	SwapInfo						:INT;
	VacValve_V8					:BOOL;	//白墨负压阀
	PurValve_V7					:BOOL;//正压阀
	alternate_Pumping		:BOOL;//交替加墨
	Swapping_Done			:BOOL;
	Error					:BOOL;
END_VAR
VAR
	step						:INT;
	stepA,stepB1,	stepB2		:INT;
	Ton,ton7,ton10				:TON;
	
	FB_SQUARE					:FB_SQUARE;
	W,X,A,Z,Y:INT;
	cycle_r_trig1,cycle_r_trig2  :R_TRIG;      //循坏
	cycle_x1,cycle_x2				:INT;//循坏次数
	purge_F_trig:F_TRIG;
	dely_off_setoff:TON;
	dely_emstop:Tc2_Standard.TON;
	ton1:Tc2_Standard.TON;
END_VAR
VAR_IN_OUT
	initialize				:BOOL;
	swap					:BOOL;
	CYCLE					:INT;//"0:Cycle A: Swap white ink to storage ;1:Cycle B: Swap storage to white ink"
	setoff					:BOOL;
END_VAR

IF setoff OR GVL.Reset THEN 
	step:=99;
END_IF
CASE step OF 
0://waiting
	IF initialize THEN 
		step :=5;
	ELSIF swap THEN 
		step :=10;
	ELSIF setoff OR GVL.Reset THEN 
		step :=99;
	END_IF
	
(***********当状态=Idle时，错误代码等于循坏错误****************************************)
	IF  state=MUStateEnum.idle THEN 
		error_code:=Circ_normal_error;
	END_IF
(***********自复位****************************************)	
	ton1(IN:=Swapping_Done , PT:= T#1S, Q=> , ET=> );
	IF ton1.Q THEN 
		Swapping_Done:=FALSE;
	END_IF
5://OFF
	state:=MUStateEnum.off;
	error_code:=MUErrorEnum.no_error;
	stepA:=stepB1:=stepB2:=0;
	W:=X:=A:=Z:=Y:=0;
	SwapInfo:=SwapInfoEnum.NONE;
	dely_emstop(IN:=FALSE);

	VacValve_V8:=FALSE;
	PurValve_V7:=FALSE;	
	
	GVL.fill_W_in_swap_enable:=FALSE;
	GVL.fill_F_in_swap_enable:=FALSE;
	
		IF initialize THEN //idle,此状态，所有泵停止	
			initialize:=FALSE;
			state:=MUStateEnum.idle;					
			GVL.fill_W_in_swap_enable:=FALSE;
			step:=0;
		END_IF
10://idle,此状态，所有泵停止				
		IF swap THEN 
			swap:=FALSE;
			state:=MUStateEnum.swapping;
			error_code:=MUErrorEnum.no_error;
			step:=20;
		END_IF
		
		IF error_code<>0 THEN 			
			step:=100;
		END_IF

20://SWAPPING		
		IF CYCLE=0 THEN
			ACT_Cycle_A();			
		ELSIF CYCLE=1 THEN 
			ACT_Cycle_B1();	
		END_IF
		
		IF SwapInfo=SwapInfoEnum.AC_STORAGE_FLUSH_FINISHED OR 
			SwapInfo=SwapInfoEnum.AC_WHITE_INK_FINISHED THEN 
			stepA:=stepB1:=stepB2:=0;		
			Swapping_Done:=TRUE;
			state:=MUStateEnum.idle;
			step:=0;
		END_IF
99://setoff
	setoff :=FALSE;
	error:=FALSE;
	state:=MUStateEnum.off;
	error_code:=MUErrorEnum.no_error;
	stepA:=stepB1:=stepB2:=0;
	W:=X:=A:=Z:=Y:=0;
	SwapInfo:=SwapInfoEnum.NONE;
	dely_emstop(IN:=FALSE);
	VacValve_V8:=FALSE;
	PurValve_V7:=FALSE;	
	
	GVL.fill_W_in_swap_enable:=FALSE;
	GVL.fill_F_in_swap_enable:=FALSE;
	step:=0;
100://error
		error:=TRUE;
		state:=MUStateEnum.error;
		stepA:=stepB1:=stepB2:=0;
		W:=X:=A:=Z:=Y:=0;
		dely_emstop(IN:=FALSE);
		VacValve_V8:=FALSE;
		PurValve_V7:=FALSE;	
		
		GVL.fill_W_in_swap_enable:=FALSE;
		GVL.fill_F_in_swap_enable:=FALSE;		
		step:=0;
END_CASE

IF setoff OR GVL.Reset THEN 
	step:=99;
END_IF

dely_off_setoff(IN:=setoff , PT:=T#1S , Q=> , ET=> );
IF dely_off_setoff.Q THEN
	setoff:=FALSE;
END_IF

IF state<>MUStateEnum.off AND state<>MUStateEnum.error  THEN 
	IF GVL.Emstop_Button THEN 
		error:=TRUE;
		error_code:=MUErrorEnum.emergency_error;
		PurValve_V7:=FALSE;
		dely_emstop(IN:=TRUE , PT:=T#1S , Q=> , ET=> );
		IF dely_emstop.Q THEN 
			VacValve_V8:=FALSE;
			step:=100;
		END_IF
	END_IF
END_IF

ACTION ACT_Cycle_A:
(***************Swap from White Ink to Storage Flush*******************************************)
CASE StepA OF
0:
	SwapInfo:=SwapInfoEnum.AC_STORAGE_FLUSH_RUNS;
	Ton(IN:=FALSE );	
	VacValve_V8:=FALSE;
	PurValve_V7 :=FALSE;
	stepA:=10;
10://SET "Vac White" OFF (valve 8 ON) 
	//START Pressure Purge Time = T1 (valve 7 ON)
	VacValve_V8:=TRUE;
	PurValve_V7 :=TRUE;
	Ton(IN:=TRUE , PT:=LREAL_TO_TIME(T[1]*1000) , Q=> , ET=> );
	IF Ton.Q THEN 
		Ton(IN:=FALSE );	
		stepA:=20;
	END_IF
20://STOP Pressure purge (normal filling conditions) (valve 7 OFF)	
	PurValve_V7:=FALSE;
	stepA:=30;
30://START Sol. filling (alternating pump time: T2=ON, T3=OFF)
	//WAIT UNTIL sensors in both TOP Sub Ink tanks detect a full tank (sensor 1 and 4)
	GVL.fill_F_in_swap_enable:=TRUE;
	alternate_Pumping:=TRUE;

	IF Sensor1 AND Sensor4 THEN 
		stepA:=31;
	END_IF
31://Wait Time: T4 (no vacuum)
	GVL.fill_F_in_swap_enable:=FALSE;
	alternate_Pumping:=FALSE;
	Ton(IN:=TRUE , PT:=LREAL_TO_TIME(T[4]*1000) , Q=> , ET=> );
		IF Ton.Q THEN 
			Ton(IN:=FALSE );
			stepA:=40;
		END_IF
40://Set "Vac White" ON  (Valve 8 OFF)     
	//Wait Time: T5 (filling conditions on & vac On)	
	VacValve_V8:=FALSE;	
	Ton(IN:=TRUE , PT:=LREAL_TO_TIME(T[5]*1000) , Q=> , ET=> );
	//调用加墨FB
		GVL.fill_F_in_swap_enable:=TRUE;
	IF Ton.Q THEN 
		stepA:=41;
	END_IF
41:
		GVL.fill_F_in_swap_enable:=FALSE;
		Ton(IN:=FALSE);
		stepA:=50;
50://Set "Vac White" Off (valve 8 ON)
	//For W=1 to 5 "Repeat 5x"
	//Pressure purge On for Time T6 (valve 7 ON)
	//Pressure purge Off for Time T6 (valve 7 OFF)
	VacValve_V8:=TRUE;
	FB_SQUARE(T_ON:=T[6] , T_OFF:=T[6] , SQUARE=>PurValve_V7 );
	purge_F_trig(CLK:=PurValve_V7 , Q=> );
	IF purge_F_trig.Q THEN 
		W:=W+1;
	END_IF
	
	IF W=6  THEN
		W:=0; 
		stepA:=60;
	END_IF
60://Wait  Time: T7 (while filling is ON)	
	Ton(IN:=TRUE  , PT:= LREAL_TO_TIME(T[7]*1000), Q=> , ET=> );	
	//调用加墨FB
	GVL.fill_F_in_swap_enable:=TRUE;
	IF ton.Q THEN 
		stepA:=61;
	END_IF
61:
		GVL.fill_F_in_swap_enable:=FALSE;
		Ton(IN:=FALSE);
		stepA:=70;
70://Set "Vac White" ON  (Valve 8 OFF)     
	//Wait Time: T5 (filling conditions on & vac On)
	VacValve_V8:=FALSE;
	//调用加墨FB
	GVL.fill_F_in_swap_enable:=TRUE;
	Ton(IN:=TRUE  , PT:= LREAL_TO_TIME(T[5]*1000), Q=> , ET=> );	
	IF ton.Q THEN 
		stepA:=71;
	END_IF
71:
		GVL.fill_F_in_swap_enable:=FALSE;
		Ton(IN:=FALSE);
		stepA:=80;
80://Set "Vac White" Off (valve 8 ON)
	VacValve_V8:=TRUE;
	//For X=1 to 5 "Repeat 5x"
	//Pressure purge On for Time T6 (valve 7 ON)
	//Pressure purge Off for Time T6 (valve 7 OFF)
	FB_SQUARE(T_ON:=T[6] , T_OFF:=T[6] , SQUARE=>PurValve_V7 );
	purge_F_trig(CLK:=PurValve_V7 , Q=> );
	IF purge_F_trig.Q THEN 
		X:=X+1;
	END_IF
	IF X=6  THEN 
		X:=0;
		stepA:=89;
	END_IF
89:
	A:=A+1;	
	stepA:=90;
90://Wait  Time: T7 (while filling is ON),第二次是T8	
	IF A<2 THEN 
		Ton(IN:=TRUE  , PT:= LREAL_TO_TIME(T[7]*1000), Q=> , ET=> );	
	ELSIF A=2 THEN 
		Ton(IN:=TRUE  , PT:= LREAL_TO_TIME(T[8]*1000), Q=> , ET=> );	
	END_IF
		//调用加墨FB
	GVL.fill_F_in_swap_enable:=TRUE;
	IF ton.Q THEN 
		stepA:=91;
	END_IF
91:
		GVL.fill_F_in_swap_enable:=FALSE;
		Ton(IN:=FALSE);
		stepA:=100;
100://Set "Vac White" ON  (Valve 8 OFF)    
	//Wait Time: T9 (filling conditions on) 
	VacValve_V8:=FALSE;
	//调用加墨FB
	GVL.fill_F_in_swap_enable:=TRUE;
	Ton(IN:=TRUE  , PT:= LREAL_TO_TIME(T[9]*1000), Q=> , ET=> );	
	IF ton.Q THEN 
		stepA:=101;
	END_IF	
101:
		GVL.fill_F_in_swap_enable:=FALSE;
		Ton(IN:=FALSE);
		stepA:=110;
110://重复	
	IF A<2 THEN 
		stepA:=10;
	ELSE stepA:=120;
	END_IF
120:(*FOR Z=1 to 5
	  IF both circulation pumps (3 & 6) were activated 3x within time: T13 => JUMP TO FINISH
	  ELSE Set Vac White Off (valve 8 ON)		
		NEXT Z*)
	A:=0;
	//	//调用加墨FB
	GVL.fill_F_in_swap_enable:=TRUE;
	Ton(IN:=TRUE  , PT:= LREAL_TO_TIME(T[13]*1000), Q=> , ET=> );	
	cycle_r_trig1(CLK:=Circ_Pump_L, Q=> );
	cycle_r_trig2(CLK:=Circ_Pump_R , Q=> );
		IF cycle_r_trig1.Q THEN 
			cycle_x1:=cycle_x1+1;
		END_IF
		IF cycle_r_trig2.Q THEN 
			cycle_x2:=cycle_x2+1;
		END_IF
		
	IF NOT Ton.Q AND cycle_x1>=3 AND cycle_x2>=3 THEN 
		Ton(IN:=FALSE);
		cycle_x1:=cycle_x2:=0;
		Z:=0;
		stepA:=190;
	ELSIF Ton.Q AND (cycle_x1<3 OR cycle_x2<3)  AND Z<5 THEN 	//循坏次数不够	
		Ton(IN:=FALSE);
		VacValve_V8:=TRUE;
		PurValve_V7:=TRUE;	
		cycle_x1:=cycle_x2:=0;
		stepA:=130;
	ELSIF Z=5 THEN
		Ton(IN:=FALSE);
		Z:=0; 
		stepA:=160;	
	END_IF
130://Start Pressure Purge On (valve 7 ON) for Time: T10
	//STOP Pressure purge (valve 7 OFF)   
			ton(IN:=TRUE , PT:= LREAL_TO_TIME(T[10]*1000) , Q=> , ET=> );		
			IF ton.Q THEN
				 ton(IN:=FALSE);
				PurValve_V7:=FALSE;
				stepA:=140;
			END_IF
140://Wait  Time: T7
		//Set "Vac White" ON  (Valve 8 OFF) 
			ton(IN:=TRUE , PT:= LREAL_TO_TIME(T[7]*1000) , Q=> , ET=> );
			IF Ton.Q THEN 
				ton(IN:=FALSE);
				VacValve_V8:=FALSE;		
				stepA:=150;
			END_IF
150://Wait Time: T11 (filling conditions on)
		//调用加墨FB
		ton(IN:=TRUE , PT:= LREAL_TO_TIME(T[11]*1000) , Q=> , ET=> );
			IF Ton.Q THEN 
				ton(IN:=FALSE);
				VacValve_V8:=FALSE;		
				Z:=Z+1;
				stepA:=120;
			END_IF
160://START WAIT = Message 2 on GUI 
	//If "PURGE BUTTON" is pushed during WAIT, THEN  
   //Set "Vac White" Off (valve 8 ON)
   //START Pressure purge (valve 7 ON) until button released
		SwapInfo:=SwapInfoEnum.AC_STORAGE_FLUSH_NEEDS_HELP;
			VacValve_V8:=TRUE;
		IF btPurge THEN 			
			PurValve_V7:=TRUE;
			stepA:=170;
		END_IF
170:    //START Pressure purge (valve 7 ON) until button released
		IF NOT btPurge THEN 
			PurValve_V7:=FALSE;
			stepA:=171;
		END_IF
171://Wait  Time: T7
	//Set "Vac White" ON  (Valve 8 OFF)  
		ton(IN:=TRUE , PT:= LREAL_TO_TIME(T[7]*1000) , Q=> , ET=> );
			IF Ton.Q THEN 
				ton(IN:=FALSE);
				VacValve_V8:=FALSE;
				stepA:=180;
			END_IF
180://  IF both circulation pumps (3 & 6) were activated 3x within time: T13 => JUMP TO FINISH
			//END IF (back TO wait)
		//	//调用加墨FB
	Ton(IN:=TRUE  , PT:= LREAL_TO_TIME(T[13]*1000), Q=> , ET=> );	
	cycle_r_trig1(CLK:=Circ_Pump_L, Q=> );
	cycle_r_trig2(CLK:=Circ_Pump_R , Q=> );
		IF cycle_r_trig1.Q THEN 
			cycle_x1:=cycle_x1+1;
		END_IF
		IF cycle_r_trig2.Q THEN 
			cycle_x2:=cycle_x2+1;
		END_IF
	IF NOT Ton.Q AND cycle_x1>=3 AND cycle_x2>=3 THEN 
		Ton(IN:=FALSE);
		cycle_x1:=cycle_x2:=0;
		stepA:=190;
	ELSIF Ton.Q AND (cycle_x1<3 OR cycle_x2<3) THEN 		
		Ton(IN:=FALSE);
		cycle_x1:=cycle_x2:=0;
		stepA:=160;
	END_IF
190:	//关闭所有供墨
	GVL.fill_F_in_swap_enable:=FALSE;
	stepA:=200;
200://FINISH => Message 3 on GUI
		SwapInfo:=SwapInfoEnum.AC_STORAGE_FLUSH_FINISHED;
		
END_CASE
END_ACTION

ACTION ACT_Cycle_B1:
(*************** Swap From Storage Flush to White Ink*******************************************)
CASE StepB1 OF
0:
	SwapInfo:=SwapInfoEnum.AC_WHITE_INK_RUNS;
	Ton(IN:=FALSE );	
	VacValve_V8:=FALSE;
	PurValve_V7 :=FALSE;
	StepB1:=10;
10://SET "Vac White" OFF (valve 8 ON) 
	//START Pressure Purge Time = T1 (valve 7 ON)
	VacValve_V8:=TRUE;
	PurValve_V7 :=TRUE;
	Ton(IN:=TRUE , PT:=LREAL_TO_TIME(T[1]*1000) , Q=> , ET=> );
	IF Ton.Q THEN 
		Ton(IN:=FALSE );	
		StepB1:=20;
	END_IF
20://STOP Pressure purge (normal filling conditions) (valve 7 OFF)	
	PurValve_V7:=FALSE;
	StepB1:=30;
30://START Ink filling  (alternating pump time: T2=ON, T3=OFF)
	//WAIT UNTIL sensors in both TOP Sub Ink tanks detect a full tank (sensor 1 and 4)	
	GVL.fill_W_in_swap_enable:=TRUE;
	alternate_Pumping:=TRUE;
	
	IF Sensor1 AND Sensor4 THEN 
		StepB1:=31;
	END_IF
31://Wait Time: T4 (no vacuum)
	GVL.fill_W_in_swap_enable:=FALSE;
	alternate_Pumping:=FALSE;
	Ton(IN:=TRUE , PT:=LREAL_TO_TIME(T[4]*1000) , Q=> , ET=> );
		IF Ton.Q THEN 
			Ton(IN:=FALSE );
			StepB1:=40;
		END_IF
40://Set "Vac White" ON  (Valve 8 OFF)     
	//Wait Time: T5 (filling conditions on & vac On)	
	VacValve_V8:=FALSE;	
	Ton(IN:=TRUE , PT:=LREAL_TO_TIME(T[5]*1000) , Q=> , ET=> );
	//调用加墨FB
		GVL.fill_W_in_swap_enable:=TRUE;
	IF Ton.Q THEN 
		StepB1:=41;
	END_IF
41:
		GVL.fill_W_in_swap_enable:=FALSE;
		Ton(IN:=FALSE);
		StepB1:=50;
50://Set "Vac White" Off (valve 8 ON)
	//For Z=1 to 5 "Repeat 5x"
	//Pressure purge On for Time T6 (valve 7 ON)
	//Pressure purge Off for Time T6 (valve 7 OFF)
	VacValve_V8:=TRUE;
	FB_SQUARE(T_ON:=T[6] , T_OFF:=T[6] , SQUARE=>PurValve_V7 );
	purge_F_trig(CLK:=PurValve_V7 , Q=> );
	IF purge_F_trig.Q THEN 
		Z:=Z+1;
	END_IF
	
	IF Z=6  THEN
		Z:=0; 
		StepB1:=60;
	END_IF
60://Wait  Time: T7
	Ton(IN:=TRUE  , PT:= LREAL_TO_TIME(T[7]*1000), Q=> , ET=> );	
	//调用加墨FB
	GVL.fill_W_in_swap_enable:=TRUE;
	IF ton.Q THEN 
		StepB1:=61;
	END_IF
61:
		GVL.fill_W_in_swap_enable:=FALSE;
		Ton(IN:=FALSE);
		StepB1:=70;
70://Set "Vac White" ON  (Valve 8 OFF)     
	//Wait Time: T5 (filling conditions on & vac On)
	VacValve_V8:=FALSE;
	//调用加墨FB
	GVL.fill_W_in_swap_enable:=TRUE;
	Ton(IN:=TRUE  , PT:= LREAL_TO_TIME(T[5]*1000), Q=> , ET=> );	
	IF ton.Q THEN 
		StepB1:=71;
	END_IF
71:
		GVL.fill_W_in_swap_enable:=FALSE;
		Ton(IN:=FALSE);
		StepB1:=80;
80://Set "Vac White" Off (valve 8 ON)
	VacValve_V8:=TRUE;
	//For Z=1 to 5 "Repeat 5x"
	//Pressure purge On for Time T6 (valve 7 ON)
	//Pressure purge Off for Time T6 (valve 7 OFF)
	FB_SQUARE(T_ON:=T[6] , T_OFF:=T[6] , SQUARE=>PurValve_V7 );
	purge_F_trig(CLK:=PurValve_V7 , Q=> );
	IF purge_F_trig.Q THEN 
		Z:=Z+1;
	END_IF
	IF Z=6  THEN 
		Z:=0;
		StepB1:=90;
	END_IF
90://Wait Time: T8 (filling conditions on, vac off))
		Ton(IN:=TRUE  , PT:= LREAL_TO_TIME(T[8]*1000), Q=> , ET=> );	
		//调用加墨FB
	GVL.fill_W_in_swap_enable:=TRUE;
	IF ton.Q THEN 
		StepB1:=91;
	END_IF
91:
		GVL.fill_W_in_swap_enable:=FALSE;
		Ton(IN:=FALSE);
		StepB1:=100;
100://Set "Vac White" ON  (Valve 8 OFF)    
	//Wait Time: T9 (filling conditions on) 
	VacValve_V8:=FALSE;
	//调用加墨FB
	GVL.fill_W_in_swap_enable:=TRUE;
	Ton(IN:=TRUE  , PT:= LREAL_TO_TIME(T[9]*1000), Q=> , ET=> );	
	IF ton.Q THEN 
		StepB1:=101;
	END_IF	
101:
		GVL.fill_W_in_swap_enable:=FALSE;
		Ton(IN:=FALSE);
		StepB1:=110;
110://无重复
		StepB1:=120;
120:(*FOR Y=1 to 5
	  IF both circulation pumps (3 & 6) were activated 3x within time: T13 => JUMP TO PAUSE
	  ELSE Set Vac White Off (valve 8 ON)		
		NEXT Y*)
	//	//调用加墨FB
	GVL.fill_W_in_swap_enable:=TRUE;
	Ton(IN:=TRUE  , PT:= LREAL_TO_TIME(T[13]*1000), Q=> , ET=> );	
	cycle_r_trig1(CLK:=Circ_Pump_L, Q=> );
	cycle_r_trig2(CLK:=Circ_Pump_R , Q=> );
		IF cycle_r_trig1.Q THEN 
			cycle_x1:=cycle_x1+1;
		END_IF
		IF cycle_r_trig2.Q THEN 
			cycle_x2:=cycle_x2+1;
		END_IF
		
	IF NOT Ton.Q AND cycle_x1>=3 AND cycle_x2>=3 THEN 
		Ton(IN:=FALSE);
		cycle_x1:=cycle_x2:=0;
		Y:=0;
		StepB1:=200;
	ELSIF Ton.Q AND (cycle_x1<3 OR cycle_x2<3)  AND Z<5 THEN 	//循坏次数不够,ELSE Set Vac White Off (valve 8 ON	
		Ton(IN:=FALSE);
		VacValve_V8:=TRUE;
		PurValve_V7:=TRUE;	
		cycle_x1:=cycle_x2:=0;
		StepB1:=130;
	ELSIF Y=5 THEN
		Ton(IN:=FALSE);
		Y:=0; 
		StepB1:=160;	
	END_IF
130://Start Pressure Purge On (valve 7 ON) for Time: T10
	//STOP Pressure purge (valve 7 OFF)   
			ton(IN:=TRUE , PT:= LREAL_TO_TIME(T[10]*1000) , Q=> , ET=> );		
			IF ton.Q THEN
				 ton(IN:=FALSE);
				PurValve_V7:=FALSE;
				StepB1:=140;
			END_IF
140://Wait  Time: T7
		//Set "Vac White" ON  (Valve 8 OFF) 
			ton(IN:=TRUE , PT:= LREAL_TO_TIME(T[7]*1000) , Q=> , ET=> );
			IF Ton.Q THEN 
				ton(IN:=FALSE);
				VacValve_V8:=FALSE;		
				StepB1:=150;
			END_IF
150://Wait Time: T11 (filling conditions on)
		//调用加墨FB
		ton(IN:=TRUE , PT:= LREAL_TO_TIME(T[11]*1000) , Q=> , ET=> );
			IF Ton.Q THEN 
				ton(IN:=FALSE);
				VacValve_V8:=FALSE;		
				Y:=Y+1;
				StepB1:=120;
			END_IF
160://START WAIT = Message 5 on GUI 
	//If "PURGE BUTTON" is pushed during WAIT, THEN  
   //Set "Vac White" Off (valve 8 ON)
   //START Pressure purge (valve 7 ON) until button released
		SwapInfo:=SwapInfoEnum.AC_WHITE_INK1_NEEDS_HELP;
			VacValve_V8:=TRUE;
		IF btPurge THEN 		
			PurValve_V7:=TRUE;
			StepB1:=170;
		END_IF
170:    //START Pressure purge (valve 7 ON) until button released
		IF NOT btPurge THEN 
			PurValve_V7:=FALSE;
			StepB1:=171;
		END_IF
171://Wait  Time: T7
	//Set "Vac White" ON  (Valve 8 OFF)  
		ton(IN:=TRUE , PT:= LREAL_TO_TIME(T[7]*1000) , Q=> , ET=> );
			IF Ton.Q THEN 
				ton(IN:=FALSE);
				VacValve_V8:=FALSE;
				StepB1:=180;
			END_IF
180://  IF both circulation pumps (3 & 6) were activated 3x within time T13 than:
		//           => remove Message 5
		//           => Show Message 4
		//           => JUMP TO PAUSE
		//END IF (back to wait)
				
		//	//调用加墨FB
	Ton(IN:=TRUE  , PT:= LREAL_TO_TIME(T[13]*1000), Q=> , ET=> );	
	cycle_r_trig1(CLK:=Circ_Pump_L, Q=> );
	cycle_r_trig2(CLK:=Circ_Pump_R , Q=> );
		IF cycle_r_trig1.Q THEN 
			cycle_x1:=cycle_x1+1;
		END_IF
		IF cycle_r_trig2.Q THEN 
			cycle_x2:=cycle_x2+1;
		END_IF
	IF NOT Ton.Q AND cycle_x1>=3 AND cycle_x2>=3 THEN 
		Ton(IN:=FALSE);
		cycle_x1:=cycle_x2:=0;
		StepB1:=190;
	ELSIF Ton.Q AND (cycle_x1<3 OR cycle_x2<3) THEN 		
		Ton(IN:=FALSE);
		cycle_x1:=cycle_x2:=0;
		StepB1:=160;
	END_IF
190:	//           => remove Message 5
		//           => Show Message 4
		//           => JUMP TO PAUSE
	SwapInfo:=SwapInfoEnum.AC_WHITE_INK_RUNS;	
	GVL.fill_W_in_swap_enable:=FALSE;
	StepB1:=200;
200://PAUSE:  wait time time: T12,Filter cleaning time
	//调用加墨FB
	GVL.fill_W_in_swap_enable:=TRUE;
	Ton(IN:=TRUE  , PT:= LREAL_TO_TIME(T[12]*1000), Q=> , ET=> );	
	IF Ton.Q THEN 
		StepB1:=210;		
	END_IF
210://关闭加墨
		Ton(IN:=FALSE);
		GVL.fill_W_in_swap_enable:=FALSE;
		StepB1:=220;
220://
	ACT_Cycle_B2();
		
END_CASE
END_ACTION

ACTION ACT_Cycle_B2:
(*************** Swap From Storage Flush to White Ink*******************************************)

CASE StepB2 OF
0:
	Ton(IN:=FALSE );	
	StepB2:=10;
10://SET "Vac White" OFF (valve 8 ON) 
	//START Pressure Purge Time = T1 (valve 7 ON)
	VacValve_V8:=TRUE;
	PurValve_V7 :=TRUE;
	Ton(IN:=TRUE , PT:=LREAL_TO_TIME(T[1]*1000) , Q=> , ET=> );
	IF Ton.Q THEN 
		Ton(IN:=FALSE );	
		StepB2:=20;
	END_IF
20://STOP Pressure purge (normal filling conditions) (valve 7 OFF)	
	PurValve_V7:=FALSE;
	StepB2:=30;
30://START Ink filling  (alternating pump time: T2=ON, T3=OFF)
	//WAIT UNTIL sensors in both TOP Sub Ink tanks detect a full tank (sensor 1 and 4)
	GVL.fill_W_in_swap_enable:=TRUE;
	alternate_Pumping:=TRUE;
	
	IF Sensor1 AND Sensor4 THEN 
		StepB2:=31;
	END_IF
31://Wait Time: T4 (no vacuum)
	GVL.fill_W_in_swap_enable:=FALSE;
	alternate_Pumping:=FALSE;
	Ton(IN:=TRUE , PT:=LREAL_TO_TIME(T[4]*1000) , Q=> , ET=> );
		IF Ton.Q THEN 
			Ton(IN:=FALSE );
			StepB2:=40;
		END_IF
40://Set "Vac White" ON  (Valve 8 OFF)     
	//Wait Time: T5 (filling conditions on & vac On)	
	VacValve_V8:=FALSE;	
	Ton(IN:=TRUE , PT:=LREAL_TO_TIME(T[5]*1000) , Q=> , ET=> );
	//调用加墨FB
		GVL.fill_W_in_swap_enable:=TRUE;
	IF Ton.Q THEN 
		StepB2:=41;
	END_IF
41:
		GVL.fill_W_in_swap_enable:=FALSE;
		Ton(IN:=FALSE);
		StepB2:=50;
50://Set "Vac White" Off (valve 8 ON)
	//For Z=1 to 5 "Repeat 5x"
	//Pressure purge On for Time T6 (valve 7 ON)
	//Pressure purge Off for Time T6 (valve 7 OFF)
	VacValve_V8:=TRUE;
	FB_SQUARE(T_ON:=T[6] , T_OFF:=T[6] , SQUARE=>PurValve_V7 );
	purge_F_trig(CLK:=PurValve_V7 , Q=> );
	IF purge_F_trig.Q THEN 
		Z:=Z+1;
	END_IF
	
	IF Z=6  THEN
		Z:=0; 
		StepB2:=60;
	END_IF
60://Wait  Time: T7
	Ton(IN:=TRUE  , PT:= LREAL_TO_TIME(T[7]*1000), Q=> , ET=> );	
	//调用加墨FB
	GVL.fill_W_in_swap_enable:=TRUE;
	IF ton.Q THEN 
		StepB2:=61;
	END_IF
61:
		GVL.fill_W_in_swap_enable:=FALSE;
		Ton(IN:=FALSE);
		StepB2:=70;
70://Set "Vac White" ON  (Valve 8 OFF)     
	//Wait Time: T5 (filling conditions on & vac On)
	VacValve_V8:=FALSE;
	//调用加墨FB
	GVL.fill_W_in_swap_enable:=TRUE;
	Ton(IN:=TRUE  , PT:= LREAL_TO_TIME(T[5]*1000), Q=> , ET=> );	
	IF ton.Q THEN 
		StepB2:=71;
	END_IF
71:
		GVL.fill_W_in_swap_enable:=FALSE;
		Ton(IN:=FALSE);
		StepB2:=80;
80://Set "Vac White" Off (valve 8 ON)
	VacValve_V8:=TRUE;
	//For Z=1 to 5 "Repeat 5x"
	//Pressure purge On for Time T6 (valve 7 ON)
	//Pressure purge Off for Time T6 (valve 7 OFF)
	FB_SQUARE(T_ON:=T[6] , T_OFF:=T[6] , SQUARE=>PurValve_V7 );
	purge_F_trig(CLK:=PurValve_V7 , Q=> );
	IF purge_F_trig.Q THEN 
		Z:=Z+1;
	END_IF
	IF Z=6  THEN 
		Z:=0;
		StepB2:=90;
	END_IF
90://Wait Time: T8 (filling conditions on, vac off))
		Ton(IN:=TRUE  , PT:= LREAL_TO_TIME(T[8]*1000), Q=> , ET=> );	
		//调用加墨FB
	GVL.fill_W_in_swap_enable:=TRUE;
	IF ton.Q THEN 
		StepB2:=91;
	END_IF
91:
		GVL.fill_W_in_swap_enable:=FALSE;
		Ton(IN:=FALSE);
		StepB2:=100;
100://Set "Vac White" ON  (Valve 8 OFF)    
	//Wait Time: T9 (filling conditions on) 
	VacValve_V8:=FALSE;
	//调用加墨FB
	GVL.fill_W_in_swap_enable:=TRUE;
	Ton(IN:=TRUE  , PT:= LREAL_TO_TIME(T[9]*1000), Q=> , ET=> );	
	IF ton.Q THEN 
		StepB2:=101;
	END_IF	
101:
		GVL.fill_W_in_swap_enable:=FALSE;
		Ton(IN:=FALSE);
		StepB2:=110;
110://无重复
		StepB2:=120;
120:(*FOR Z=1 to 5
	  IF both circulation pumps (3 & 6) were activated 3x within time: T13 => JUMP TO FINISH
	  ELSE Set Vac White Off (valve 8 ON)		
		NEXT Z*)
	//	//调用加墨FB
	GVL.fill_W_in_swap_enable:=TRUE;
	Ton(IN:=TRUE  , PT:= LREAL_TO_TIME(T[13]*1000), Q=> , ET=> );	
	cycle_r_trig1(CLK:=Circ_Pump_L, Q=> );
	cycle_r_trig2(CLK:=Circ_Pump_R , Q=> );
		IF cycle_r_trig1.Q THEN 
			cycle_x1:=cycle_x1+1;
		END_IF
		IF cycle_r_trig2.Q THEN 
			cycle_x2:=cycle_x2+1;
		END_IF
		
	IF NOT Ton.Q AND cycle_x1>=3 AND cycle_x2>=3 THEN 
		Ton(IN:=FALSE);
		cycle_x1:=cycle_x2:=0;
		Z:=0;
		StepB2:=200;
	ELSIF Ton.Q AND (cycle_x1<3 OR cycle_x2<3)  AND Z<5 THEN 	//循坏次数不够,ELSE Set Vac White Off (valve 8 ON	
		Ton(IN:=FALSE);
		VacValve_V8:=TRUE;
		PurValve_V7:=TRUE;	
		cycle_x1:=cycle_x2:=0;
		StepB2:=130;
	ELSIF Z=5 THEN
		Ton(IN:=FALSE);
		Z:=0; 
		StepB2:=160;	
	END_IF
130://Start Pressure Purge On (valve 7 ON) for Time: T10
	//STOP Pressure purge (valve 7 OFF)   
			ton(IN:=TRUE , PT:= LREAL_TO_TIME(T[10]*1000) , Q=> , ET=> );		
			IF ton.Q THEN
				 ton(IN:=FALSE);
				PurValve_V7:=FALSE;
				StepB2:=140;
			END_IF
140://Wait  Time: T7
		//Set "Vac White" ON  (Valve 8 OFF) 
			ton(IN:=TRUE , PT:= LREAL_TO_TIME(T[7]*1000) , Q=> , ET=> );
			IF Ton.Q THEN 
				ton(IN:=FALSE);
				VacValve_V8:=FALSE;		
				StepB2:=150;
			END_IF
150://Wait Time: T11 (filling conditions on)
		//调用加墨FB
		ton(IN:=TRUE , PT:= LREAL_TO_TIME(T[11]*1000) , Q=> , ET=> );
			IF Ton.Q THEN 
				ton(IN:=FALSE);
				VacValve_V8:=FALSE;		
				Z:=Z+1;
				StepB2:=120;
			END_IF
160://START WAIT = Message 6 on GUI 
	//If "PURGE BUTTON" is pushed during WAIT, THEN  
   //Set "Vac White" Off (valve 8 ON)
   //START Pressure purge (valve 7 ON) until button released
		SwapInfo:=SwapInfoEnum.AC_WHITE_INK2_NEEDS_HELP;
			VacValve_V8:=TRUE;
		IF btPurge THEN 			
			PurValve_V7:=TRUE;
			StepB2:=170;
		END_IF
170:    //START Pressure purge (valve 7 ON) until button released
		IF NOT btPurge THEN 
			PurValve_V7:=FALSE;
			StepB2:=171;
		END_IF
171://Wait  Time: T7
	//Set "Vac White" ON  (Valve 8 OFF)  
		ton(IN:=TRUE , PT:= LREAL_TO_TIME(T[7]*1000) , Q=> , ET=> );
			IF Ton.Q THEN 
				ton(IN:=FALSE);
				VacValve_V8:=FALSE;
				StepB2:=180;
			END_IF
180://    IF both circulation pumps (3 & 6) were activated 3x within time: T13 => JUMP TO FINISH
		//END IF (back to wait)
				
		//	//调用加墨FB
	Ton(IN:=TRUE  , PT:= LREAL_TO_TIME(T[13]*1000), Q=> , ET=> );	
	cycle_r_trig1(CLK:=Circ_Pump_L, Q=> );
	cycle_r_trig2(CLK:=Circ_Pump_R , Q=> );
		IF cycle_r_trig1.Q THEN 
			cycle_x1:=cycle_x1+1;
		END_IF
		IF cycle_r_trig2.Q THEN 
			cycle_x2:=cycle_x2+1;
		END_IF
	IF NOT Ton.Q AND cycle_x1>=3 AND cycle_x2>=3 THEN 
		Ton(IN:=FALSE);
		cycle_x1:=cycle_x2:=0;
		StepB2:=190;
	ELSIF Ton.Q AND (cycle_x1<3 OR cycle_x2<3) THEN 		
		Ton(IN:=FALSE);
		cycle_x1:=cycle_x2:=0;
		StepB2:=160;
	END_IF
190:	//  
	StepB2:=200;
200://
	StepB2:=210;
210://关闭加墨
	Ton(IN:=FALSE);
	GVL.fill_W_in_swap_enable:=FALSE;
	StepB2:=220;
220://FINISH => Message 7 on GUI
	SwapInfo:=SwapInfoEnum.AC_WHITE_INK_FINISHED;

		
END_CASE
END_ACTION

END_FUNCTION_BLOCK

// ---- POUs/MAIN.TcPOU
PROGRAM MAIN
VAR
	FB_count:FB_count;
END_VAR

P_UPS();
systime();

IO_Link();
P_API_IO();
P_Modbus();
MAIN_ALarm();

P_Motion();
P_MediaTransport();
P_System();
P_InkSystem();
P_UVLed();
P_RollToRoll();
P_SpitUnit();
P_MaintenanceUnit();
P_SubTank();
P_TwinSAFE();


ACT_heart();



//IF VisuElems.CURRENTVISU='VIS_AXIS' THEN 
	//VisuElems.CURRENTVISU:='VIS_ISS';
//END_IF

ACTION ACT_heart:
FB_count(Add_Time:=T#0.1S , count=> GVL_API.count );
END_ACTION

END_PROGRAM

// ---- POUs/040_System/P_System.TcPOU
PROGRAM P_System
VAR
END_VAR

P_FootPedal();
P_SystemEnvironment();
P_SafetyGuard();

END_PROGRAM

// ---- POUs/040_System/FootPedal/P_FootPedal.TcPOU
PROGRAM P_FootPedal
VAR
	FB_FootPedal:ARRAY[1..number_FootPedal] OF FB_FootPedal;//
	i:INT;
	log_ErrorEnum:FootPedalErrorEnum;
	log_ID:INT;
END_VAR

ACT_LOG();
FOR i:=1 TO number_FootPedal DO
	FB_FootPedal[i](
		PedalPressed1:=stInput.biFootPedal[i].PedalPressed1 , 
		PedalPressed2:=stInput.biFootPedal[i].PedalPressed2 , 
		PedalPressed3:=stInput.biFootPedal[i].PedalPressed3 , 
		debounce_time:=GVL_API.stFootPedal[i].debounce_time , 
		error_code=> GVL_API.stFootPedal[i].error_code, 
		state=> GVL_API.stFootPedal[i].state, 
		pressed=> GVL_API.stFootPedal[i].pressed, 
		Error=>GVL_API.stFootPedal[i].Error , 
		Reset:= GVL_API.stFootPedal[i].Reset );
END_FOR

ACTION ACT_LOG:
(*************************LOG*******************************************)
log_ID:=400;
FOR i:=1 TO number_FootPedal DO//401-404
//pressed
AlarmActionArray[log_ID+i].AlarmMsg.EN	:=CONCAT('FootPedal',
																			INT_TO_STRING(i));
AlarmActionArray[log_ID+i].AlarmMsg.EN	:=CONCAT(AlarmActionArray[log_ID+i].AlarmMsg.EN,': '	);																	
AlarmActionArray[log_ID+i].AlarmMsg.EN	:=CONCAT(AlarmActionArray[log_ID+i].AlarmMsg.EN,
																			INT_TO_STRING(GVL_API.stFootPedal[i].pressed));												
fbSetAlarm[log_ID+i](
	InUse:=TRUE , 
	EventId:=log_ID+i , 
	EventActive:=GVL_API.stFootPedal[i].pressed<>0 , 
	EventClass:=Alm_EventClass.Event , 
	ToTheLogFile:=TRUE, 
	ToTheHistory:=TRUE , 
 );
 
//ERROR,log_ErrorEnum只能等于一个常数,   410-414
CASE GVL_API.stUpDownSlot[i].error_code  OF
0	:	log_ErrorEnum	:=	0	;
1	:	log_ErrorEnum	:=	1	;
2	:	log_ErrorEnum	:=	2	;
3	:	log_ErrorEnum	:=	3	;
4	:	log_ErrorEnum	:=	4	;
666	:	log_ErrorEnum	:=	666	;


END_CASE
AlarmActionArray[log_ID+10+i].AlarmMsg.EN	:=CONCAT('FootPedal',INT_TO_STRING(i));
AlarmActionArray[log_ID+10+i].AlarmMsg.EN	:=CONCAT(AlarmActionArray[log_ID+10+i].AlarmMsg.EN,
																			' Error: ');
AlarmActionArray[log_ID+10+i].AlarmMsg.EN	:=CONCAT(AlarmActionArray[log_ID+10+i].AlarmMsg.EN,
																			TO_STRING(log_ErrorEnum));																			

fbSetAlarm[log_ID+10+i](
	InUse:=TRUE , 
	EventId:=log_ID+10+i , 
	EventActive:=GVL_API.stFootPedal[i].error_code<>0 AND GVL_API.stFootPedal[i].error_code<>666  , 
	EventClass:=Alm_EventClass.Alarm , 
	ToTheLogFile:=TRUE, 
	ToTheHistory:=TRUE , 
 );
 
//reset  420-424
AlarmActionArray[log_ID+20+i].AlarmMsg.EN	:=CONCAT('FootPedal',
																			INT_TO_STRING(i));
AlarmActionArray[log_ID+20+i].AlarmMsg.EN	:=CONCAT(AlarmActionArray[log_ID+20+i].AlarmMsg.EN,
																			' Reset');		

fbSetAlarm[log_ID+20+i](
	InUse:=TRUE , 
	EventId:=log_ID+20+i , 
	EventActive:=GVL_API.stFootPedal[i].Reset  , 
	EventClass:=Alm_EventClass.Event , 
	ToTheLogFile:=TRUE, 
	ToTheHistory:=TRUE , 
 );
END_FOR
END_ACTION

END_PROGRAM

// ---- POUs/060_UVLed/P_UVLed.TcPOU
PROGRAM P_UVLed
VAR
	//FB_UVLed		:FB_UVLed;
	FB_UVLed_L		:FB_UVLed_L;
	FB_UVLed_R		:FB_UVLed_R;

	log_ErrorEnum:UVLedErrorEnum;
	log_ID:INT;
	i:INT;
END_VAR

ACT_LOG();
FB_UVLed_L(
	single_double:=GVL_API.stUVLed[1].unidirection , 
	initial_print_position:= GVL_API.stUVLed[1].initial_print_position, 
	uv_power_leading:= GVL_API.stUVLed[1].uv_power_leading, 
	uv_power_trailing:= GVL_API.stUVLed[1].uv_power_trailing, 
	uvStart:= GVL_API.stUVLed[1].uvStart, 
	uvEnd:= GVL_API.stUVLed[1].uvEnd,
	ahead_pos:=GVL_API.stUVLed[1].ahead_pos,
	delay_pos:=GVL_API.stUVLed[1].delay_pos, 
	parts:=GVL_API.stUVLed[1].prats,
	Encoder:= Axis[FastScan].Ref.NcToPlc.ActPos, 
	Moving:= Axis[FastScan].Ref.Status.Moving, 
	FS_Direction_N:= Axis[FastScan].Ref.Status.NegativeDirection, 
	FS_Direction_P:=Axis[FastScan].Ref.Status.PositiveDirection , 	
	UVError:=GVL.UV_error_L , 
	//IO_Error:=GVL.UV_timeout,
	UVisRemote:=GVL.UVisRemote,
	state=> GVL_API.stUVLed[1].state, 
	error_code=> GVL_API.stUVLed[1].error_code, 
	uv_power=>GVL.set_uv_power_left, 
	set_prats=>GVL.set_uv_parts_left,
	initialized=> GVL_API.stUVLed[1].initialized, 
	settings_applide=>GVL_API.stUVLed[1].settings_applied , 
	curing_started=> GVL_API.stUVLed[1].curing_started, 
	curing_stopped=> GVL_API.stUVLed[1].curing_stopped, 
	error=> GVL_API.stUVLed[1].error, 
	off=> GVL_API.stUVLed[1].off,
	Initialize:= GVL_API.stUVLed[1].Initialize, 
	ConfigurePowerSettings:= GVL_API.stUVLed[1].ConfigurePowerSettings, 
	ConfigurePositions:= GVL_API.stUVLed[1].ConfigurePositions, 
	StopCuring:= GVL_API.stUVLed[1].StopCuring, 
	SetOff:=GVL_API.stUVLed[1].SetOff  );
FB_UVLed_R(
	single_double:=GVL_API.stUVLed[2].unidirection , 
	initial_print_position:= GVL_API.stUVLed[2].initial_print_position, 
	uv_power_leading:= GVL_API.stUVLed[2].uv_power_leading, 
	uv_power_trailing:= GVL_API.stUVLed[2].uv_power_trailing, 
	uvStart:= GVL_API.stUVLed[2].uvStart, 
	uvEnd:= GVL_API.stUVLed[2].uvEnd, 
	ahead_pos:=GVL_API.stUVLed[2].ahead_pos,
	delay_pos:=GVL_API.stUVLed[2].delay_pos,
	parts:=GVL_API.stUVLed[2].prats,
	Encoder:= Axis[FastScan].Ref.NcToPlc.ActPos, 
	Moving:= Axis[FastScan].Ref.Status.Moving, 
	FS_Direction_N:= Axis[FastScan].Ref.Status.NegativeDirection, 
	FS_Direction_P:=Axis[FastScan].Ref.Status.PositiveDirection , 
	UVError:=GVL.UV_error_R ,
	//IO_Error:=GVL.UV_timeout, 
	UVisRemote:=GVL.UVisRemote,
	state=> GVL_API.stUVLed[2].state, 
	error_code=> GVL_API.stUVLed[2].error_code, 
	uv_power=>GVL. set_uv_power_right, 
	set_prats=>GVL.set_uv_parts_right,
	initialized=> GVL_API.stUVLed[2].initialized, 
	settings_applide=>GVL_API.stUVLed[2].settings_applied , 
	curing_started=> GVL_API.stUVLed[2].curing_started, 
	curing_stopped=> GVL_API.stUVLed[2].curing_stopped, 
	error=> GVL_API.stUVLed[2].error, 
	off=> GVL_API.stUVLed[2].off,
	Initialize:= GVL_API.stUVLed[2].Initialize, 
	ConfigurePowerSettings:= GVL_API.stUVLed[2].ConfigurePowerSettings, 
	ConfigurePositions:= GVL_API.stUVLed[2].ConfigurePositions, 
	StopCuring:= GVL_API.stUVLed[2].StopCuring, 
	SetOff:=GVL_API.stUVLed[2].SetOff  );

ACTION ACT_LOG:
(*************************LOG*******************************************)
log_ID:=600;

FOR i:=1 TO 2 DO 
(*uv1:500-549    uv2:550-   *)
//initialize
AlarmActionArray[log_ID+50*i-50+1].AlarmMsg.EN	:=	CONCAT('UVLed',INT_TO_STRING(i));
AlarmActionArray[log_ID+50*i-50+1].AlarmMsg.EN	:=	CONCAT(AlarmActionArray[log_ID+50*i-50+1].AlarmMsg.EN,
																				' Initialize');

fbSetAlarm[log_ID+50*i-50+1](
	InUse:=TRUE , 
	EventId:=log_ID+50*i-50+1 , 
	EventActive:=GVL_API.stUVLed[i].Initialize , 
	EventClass:=Alm_EventClass.Event , 
	ToTheLogFile:=TRUE, 
	ToTheHistory:=TRUE , 
 );

 //ConfigurePowerSettings
AlarmActionArray[log_ID+50*i-50+2].AlarmMsg.EN	:=	CONCAT('UVLed',INT_TO_STRING(i));
AlarmActionArray[log_ID+50*i-50+2].AlarmMsg.EN	:=	CONCAT(AlarmActionArray[log_ID+50*i-50+2].AlarmMsg.EN,
																				' ConfigurePowerSettings: ');
	IF GVL_API.stUVLed[i].initial_print_position=0 THEN 
	AlarmActionArray[log_ID+50*i-50+2].AlarmMsg.EN	:=	CONCAT(AlarmActionArray[log_ID+50*i-50+2].AlarmMsg.EN,
																					'from_home;');
	ELSE 
	AlarmActionArray[log_ID+50*i-50+2].AlarmMsg.EN	:=	CONCAT(AlarmActionArray[log_ID+50*i-50+2].AlarmMsg.EN,
																					'to_home;');																			
	END_IF
 	IF GVL_API.stUVLed[i].unidirection THEN 
	AlarmActionArray[log_ID+50*i-50+2].AlarmMsg.EN	:=	CONCAT(AlarmActionArray[log_ID+50*i-50+2].AlarmMsg.EN,
																					'bi-directional;');	
	ELSE
	AlarmActionArray[log_ID+50*i-50+2].AlarmMsg.EN	:=	CONCAT(AlarmActionArray[log_ID+50*i-50+2].AlarmMsg.EN,
																					'unidirectional;');	
	END_IF
	AlarmActionArray[log_ID+50*i-50+2].AlarmMsg.EN	:=	CONCAT(AlarmActionArray[log_ID+50*i-50+2].AlarmMsg.EN,
																					DINT_TO_STRING(GVL_API.stUVLed[i].uv_power_leading));	
	AlarmActionArray[log_ID+50*i-50+2].AlarmMsg.EN	:=	CONCAT(AlarmActionArray[log_ID+50*i-50+2].AlarmMsg.EN,';');
	AlarmActionArray[log_ID+50*i-50+2].AlarmMsg.EN	:=	CONCAT(AlarmActionArray[log_ID+50*i-50+2].AlarmMsg.EN,
																					DINT_TO_STRING(GVL_API.stUVLed[i].uv_power_trailing));	
fbSetAlarm[log_ID+50*i-50+2](
	InUse:=TRUE , 
	EventId:=log_ID+50*i-50+2 , 
	EventActive:=GVL_API.stUVLed[i].ConfigurePowerSettings , 
	EventClass:=Alm_EventClass.Event , 
	ToTheLogFile:=TRUE, 
	ToTheHistory:=TRUE , 
 );	
//ConfigurePositions
AlarmActionArray[log_ID+50*i-50+3].AlarmMsg.EN	:=	CONCAT('UVLed',INT_TO_STRING(i));
AlarmActionArray[log_ID+50*i-50+3].AlarmMsg.EN	:=	CONCAT(AlarmActionArray[log_ID+50*i-50+3].AlarmMsg.EN,
																				' ConfigurePositions: ');
AlarmActionArray[log_ID+50*i-50+3].AlarmMsg.EN	:=	CONCAT(AlarmActionArray[log_ID+50*i-50+3].AlarmMsg.EN,
																					LREAL_TO_STRING(GVL_API.stUVLed[i].uvStart));	
AlarmActionArray[log_ID+50*i-50+3].AlarmMsg.EN	:=	CONCAT(AlarmActionArray[log_ID+50*i-50+3].AlarmMsg.EN,',');	
AlarmActionArray[log_ID+50*i-50+3].AlarmMsg.EN	:=	CONCAT(AlarmActionArray[log_ID+50*i-50+3].AlarmMsg.EN,
																					LREAL_TO_STRING(GVL_API.stUVLed[i].uvEnd));
																					
fbSetAlarm[log_ID+50*i-50+3](
	InUse:=TRUE , 
	EventId:=log_ID+50*i-50+3 , 
	EventActive:=GVL_API.stUVLed[i].ConfigurePositions , 
	EventClass:=Alm_EventClass.Event , 
	ToTheLogFile:=TRUE, 
	ToTheHistory:=TRUE , 
);	
//StopCuring
AlarmActionArray[log_ID+50*i-50+4].AlarmMsg.EN	:=	CONCAT('UVLed',INT_TO_STRING(i));
AlarmActionArray[log_ID+50*i-50+4].AlarmMsg.EN	:=	CONCAT(AlarmActionArray[log_ID+50*i-50+4].AlarmMsg.EN,
																				' StopCuring');
																				
fbSetAlarm[log_ID+50*i-50+4](
	InUse:=TRUE , 
	EventId:=log_ID+50*i-50+4 , 
	EventActive:=GVL_API.stUVLed[i].StopCuring , 
	EventClass:=Alm_EventClass.Event , 
	ToTheLogFile:=TRUE, 
	ToTheHistory:=TRUE , 
);	
//ERROR,log_ErrorEnum只能等于一个常数
CASE GVL_API.stUVLed[i].error_code OF
0	:	log_ErrorEnum	:=	0	;
1	:	log_ErrorEnum	:=	1	;
2	:	log_ErrorEnum	:=	2	;
3	:	log_ErrorEnum	:=	3	;
4	:	log_ErrorEnum	:=	4	;
666	:	log_ErrorEnum	:=	666	;
END_CASE

AlarmActionArray[log_ID+50*i-50+5].AlarmMsg.EN	:=	CONCAT('UVLed',INT_TO_STRING(i));
AlarmActionArray[log_ID+50*i-50+5].AlarmMsg.EN	:=	CONCAT(AlarmActionArray[log_ID+50*i-50+5].AlarmMsg.EN,
																				' Error: ');
AlarmActionArray[log_ID+50*i-50+5].AlarmMsg.EN	:=	CONCAT(AlarmActionArray[log_ID+50*i-50+5].AlarmMsg.EN,
																				TO_STRING(log_ErrorEnum));

fbSetAlarm[log_ID+50*i-50+5](
	InUse:=TRUE , 
	EventId:=log_ID+50*i-50+5 , 
	EventActive:=GVL_API.stUVLed[i].error_code<>0 AND GVL_API.stUVLed[i].error_code<>666 , 
	EventClass:=Alm_EventClass.Alarm , 
	ToTheLogFile:=TRUE, 
	ToTheHistory:=TRUE , 
 );		

//SetOff
AlarmActionArray[log_ID+50*i-50+6].AlarmMsg.EN	:=	CONCAT('UVLed',INT_TO_STRING(i));
AlarmActionArray[log_ID+50*i-50+6].AlarmMsg.EN	:=	CONCAT(AlarmActionArray[log_ID+50*i-50+6].AlarmMsg.EN,
																				' SetOff: ');
																				
fbSetAlarm[log_ID+50*i-50+6](
	InUse:=TRUE , 
	EventId:=log_ID+50*i-50+6 , 
	EventActive:=GVL_API.stUVLed[i].SetOff , 
	EventClass:=Alm_EventClass.Alarm , 
	ToTheLogFile:=TRUE, 
	ToTheHistory:=TRUE , 
 );		
															
END_FOR
 (*************em-stop*     680*************
AlarmActionArray[680].AlarmMsg.EN	:=	'UVLed Error: emergency_error';
fbSetAlarm[680](
	InUse:=TRUE , 
	EventId:=680 , 
	EventActive:=GVL_API.stUVLed[1].error_code=666 OR  GVL_API.stUVLed[2].error_code=666, 
	EventClass:=Alm_EventClass.Alarm , 
	ToTheLogFile:=TRUE, 
	ToTheHistory:=TRUE , 
 );		
*)
END_ACTION

END_PROGRAM

// ---- POUs/070_RollToRoll/P_RollToRoll.TcPOU
PROGRAM P_RollToRoll
VAR
	FB_RoolToRool  :ARRAY[1..number_RoolToRool] OF FB_RollToRoll_Torque;//  1:input1; 2:output1; 3:input2; 4:output2  
 	single_double:BOOL;//1:double;0:single
	i:INT;
	log_ErrorEnum:RTRErrorEnum;
	log_ID:INT;
	
	old_usable:BOOL;
	ton_old_usable:Tc2_Standard.TON;
	
	old_isprinting:BOOL;
	ton_old_isprinting:Tc2_Standard.TON;
	
	Max_profile_velocity AT%Q*:ARRAY[1..4] OF UDINT;//转矩模式下速度限制 单位0.1r/min
END_VAR

ACT_LOG();

(*************单双卷***************************)
(*********刹车控制：单卷时，刹车同时控制**********)
IF stInput.biDualSensor[1] AND stInput.biDualSensor[2]  THEN //DOUBLE
	GVL_API.stRoolToRool[1].usable:=GVL_API.stRoolToRool[2].usable:=GVL_API.stRoolToRool[3].usable:=GVL_API.stRoolToRool[4].usable:=TRUE;
	stOutput.bqBreakPower[1]:=FB_RoolToRool[1].Break_Power;
	stOutput.bqBreakPower[3]:=FB_RoolToRool[3].Break_Power;
	single_double:=TRUE;
ELSIF NOT stInput.biDualSensor[1] AND NOT stInput.biDualSensor[2] THEN //SINGLE
	GVL_API.stRoolToRool[1].usable:=GVL_API.stRoolToRool[2].usable:=TRUE;
	GVL_API.stRoolToRool[3].usable:=GVL_API.stRoolToRool[4].usable:=FALSE;
	stOutput.bqBreakPower[1]:=FB_RoolToRool[1].Break_Power;
	stOutput.bqBreakPower[3]:=FB_RoolToRool[1].Break_Power;
	single_double:=FALSE;
ELSE
	GVL_API.stRoolToRool[1].usable:=GVL_API.stRoolToRool[2].usable:=GVL_API.stRoolToRool[3].usable:=GVL_API.stRoolToRool[4].usable:=FALSE;
END_IF

(*********速度限制**************)
FOR i:=1 TO 4 DO
	Max_profile_velocity[i]:=3000*GVL_API.stRoolToRool[i].rate/10;
END_FOR

FB_RoolToRool[1](
		biClamp_hold:=stInput.biClamp_hold[1],
		Un_Rewinder:=FALSE,
		Max_velo:=3000 , 
		REF:= , 
		usable:=GVL_API.stRoolToRool[1].usable, 
		acceleration:= GVL_API.stRoolToRool[1].acceleration, 
		deceleration:=GVL_API.stRoolToRool[1].deceleration , 
		rate:=HMI_RTR_set_Torque[1], 
		untension_rate:= GVL_API.stRoolToRool[1].untension_rate, 
		tension_mode:= GVL_API.stRoolToRool[1].tension_mode, 
		tension_timeout:= GVL_API.stRoolToRool[1].tension_timeout, 
		untension_timeout:= GVL_API.stRoolToRool[1].untension_timeout, 
		brake_timeout:= GVL_API.stRoolToRool[1].brake_timeout, 
		error_code=> GVL_API.stRoolToRool[1].error_code, 
		state=> GVL_API.stRoolToRool[1].state, 
		Axis_ErrorId=> GVL_API.stRoolToRool[1].AxisErrorId, 
		Break_Power=>  , 
		Clutch_Out=> stOutput .bqCluthOut[1], 
		Initialize:= GVL_API.stRoolToRool[1].Initialize, 
		SetActivate:= GVL_API.stRoolToRool[1].SetActivate, 
		SetReady:= GVL_API.stRoolToRool[1].SetReady, 
		EnableBrake:= GVL_API.stRoolToRool[1].EnableBrake, 
		DisableBrake:= GVL_API.stRoolToRool[1].DisableBrake, 
		StartTension:= GVL_API.stRoolToRool[1].StartTension, 
		StopTension:= GVL_API.stRoolToRool[1].StopTension, 
		Unlock:= GVL_API.stRoolToRool[1].Unlock, 
		Lock:= GVL_API.stRoolToRool[1].Lock, 
		SetOff:= GVL_API.stRoolToRool[1].SetOff ,
		Initialized=> GVL_API.stRoolToRool[1].Initialized, 
		error=> GVL_API.stRoolToRool[1].error, 
		tensioned=> GVL_API.stRoolToRool[1].tensioned, 
		untensioned=>GVL_API.stRoolToRool[1].untensioned );

FB_RoolToRool[2](
		biClamp_hold:=stInput.biClamp_hold[2],
		Un_Rewinder:=TRUE,
		Max_velo:=3000 , 
		REF:= , 		
		usable:=GVL_API.stRoolToRool[2].usable, 
		acceleration:= GVL_API.stRoolToRool[2].acceleration, 
		deceleration:=GVL_API.stRoolToRool[2].deceleration , 
		rate:= HMI_RTR_set_Torque[2], 
		untension_rate:= GVL_API.stRoolToRool[2].untension_rate, 
		tension_mode:= GVL_API.stRoolToRool[2].tension_mode, 
		tension_timeout:= GVL_API.stRoolToRool[2].tension_timeout, 
		untension_timeout:= GVL_API.stRoolToRool[2].untension_timeout, 
		brake_timeout:= GVL_API.stRoolToRool[2].brake_timeout, 
		error_code=> GVL_API.stRoolToRool[2].error_code, 
		state=> GVL_API.stRoolToRool[2].state, 
		Axis_ErrorId=> GVL_API.stRoolToRool[2].AxisErrorId, 
		Break_Power=> , 
		Clutch_Out=> stOutput .bqCluthOut[2], 
		Initialize:= GVL_API.stRoolToRool[2].Initialize, 
		SetActivate:= GVL_API.stRoolToRool[2].SetActivate, 
		SetReady:= GVL_API.stRoolToRool[2].SetReady, 
		EnableBrake:= GVL_API.stRoolToRool[2].EnableBrake, 
		DisableBrake:= GVL_API.stRoolToRool[2].DisableBrake, 
		StartTension:= GVL_API.stRoolToRool[2].StartTension, 
		StopTension:= GVL_API.stRoolToRool[2].StopTension, 
		Unlock:= GVL_API.stRoolToRool[2].Unlock, 
		Lock:= GVL_API.stRoolToRool[2].Lock, 
		SetOff:= GVL_API.stRoolToRool[2].SetOff ,
		Initialized=> GVL_API.stRoolToRool[2].Initialized, 
		error=> GVL_API.stRoolToRool[2].error, 
		tensioned=> GVL_API.stRoolToRool[2].tensioned, 
		untensioned=>GVL_API.stRoolToRool[2].untensioned);
		
FB_RoolToRool[3](
		biClamp_hold:=stInput.biClamp_hold[1],
		Un_Rewinder:=FALSE,
		Max_velo:=3000 , 
		REF:= , 
		usable:=GVL_API.stRoolToRool[3].usable, 
		acceleration:= GVL_API.stRoolToRool[3].acceleration, 
		deceleration:=GVL_API.stRoolToRool[3].deceleration , 
		rate:= HMI_RTR_set_Torque[3], 
		untension_rate:= GVL_API.stRoolToRool[3].untension_rate, 
		tension_mode:= GVL_API.stRoolToRool[3].tension_mode, 
		tension_timeout:= GVL_API.stRoolToRool[3].tension_timeout, 
		untension_timeout:= GVL_API.stRoolToRool[3].untension_timeout, 
		brake_timeout:= GVL_API.stRoolToRool[3].brake_timeout, 
		error_code=> GVL_API.stRoolToRool[3].error_code, 
		state=> GVL_API.stRoolToRool[3].state, 
		Axis_ErrorId=> GVL_API.stRoolToRool[3].AxisErrorId, 
		Break_Power=> , 
		Clutch_Out=> stOutput .bqCluthOut[3], 
		Initialize:= GVL_API.stRoolToRool[3].Initialize, 
		SetActivate:= GVL_API.stRoolToRool[3].SetActivate, 
		SetReady:= GVL_API.stRoolToRool[3].SetReady, 
		EnableBrake:= GVL_API.stRoolToRool[3].EnableBrake, 
		DisableBrake:= GVL_API.stRoolToRool[3].DisableBrake, 
		StartTension:= GVL_API.stRoolToRool[3].StartTension, 
		StopTension:= GVL_API.stRoolToRool[3].StopTension, 
		Unlock:= GVL_API.stRoolToRool[3].Unlock, 
		Lock:= GVL_API.stRoolToRool[3].Lock, 
		SetOff:= GVL_API.stRoolToRool[3].SetOff ,
		Initialized=> GVL_API.stRoolToRool[3].Initialized, 
		error=> GVL_API.stRoolToRool[3].error, 
		tensioned=> GVL_API.stRoolToRool[3].tensioned, 
		untensioned=>GVL_API.stRoolToRool[3].untensioned);
		
FB_RoolToRool[4](
		biClamp_hold:=stInput.biClamp_hold[2],
		Un_Rewinder:=TRUE,
		Max_velo:=3000 , 
		REF:= , 
		usable:=GVL_API.stRoolToRool[4].usable, 
		acceleration:= GVL_API.stRoolToRool[4].acceleration, 
		deceleration:=GVL_API.stRoolToRool[4].deceleration , 
		rate:= HMI_RTR_set_Torque[4], 
		untension_rate:= GVL_API.stRoolToRool[4].untension_rate, 
		tension_mode:= GVL_API.stRoolToRool[4].tension_mode, 
		tension_timeout:= GVL_API.stRoolToRool[4].tension_timeout, 
		untension_timeout:= GVL_API.stRoolToRool[4].untension_timeout, 
		brake_timeout:= GVL_API.stRoolToRool[4].brake_timeout, 
		error_code=> GVL_API.stRoolToRool[4].error_code, 
		state=> GVL_API.stRoolToRool[4].state, 
		Axis_ErrorId=> GVL_API.stRoolToRool[4].AxisErrorId, 
		Break_Power=> , 
		Clutch_Out=> stOutput .bqCluthOut[4], 
		Initialize:= GVL_API.stRoolToRool[4].Initialize, 
		SetActivate:= GVL_API.stRoolToRool[4].SetActivate, 
		SetReady:= GVL_API.stRoolToRool[4].SetReady, 
		EnableBrake:= GVL_API.stRoolToRool[4].EnableBrake, 
		DisableBrake:= GVL_API.stRoolToRool[4].DisableBrake, 
		StartTension:= GVL_API.stRoolToRool[4].StartTension, 
		StopTension:= GVL_API.stRoolToRool[4].StopTension, 
		Unlock:= GVL_API.stRoolToRool[4].Unlock, 
		Lock:= GVL_API.stRoolToRool[4].Lock, 
		SetOff:= GVL_API.stRoolToRool[4].SetOff ,
		Initialized=> GVL_API.stRoolToRool[4].Initialized, 
		error=> GVL_API.stRoolToRool[4].error, 
		tensioned=> GVL_API.stRoolToRool[4].tensioned, 
		untensioned=>GVL_API.stRoolToRool[4].untensioned);

ACTION ACT_LOG:
(*************************LOG*******************************************)
log_ID:=700;

FOR i:=1 TO number_RoolToRool DO //700-780
//Initialize
AlarmActionArray[log_ID+20*i-20+1].AlarmMsg.EN	:=	CONCAT('Rool-',INT_TO_STRING(i));
AlarmActionArray[log_ID+20*i-20+1].AlarmMsg.EN	:=	CONCAT(AlarmActionArray[log_ID+20*i-20+1].AlarmMsg.EN,
																				' Initialize acc:');
AlarmActionArray[log_ID+20*i-20+1].AlarmMsg.EN	:=	CONCAT(AlarmActionArray[log_ID+20*i-20+1].AlarmMsg.EN,
																				LREAL_TO_STRING(GVL_API.stRoolToRool[i].acceleration));
AlarmActionArray[log_ID+20*i-20+1].AlarmMsg.EN	:=	CONCAT(AlarmActionArray[log_ID+20*i-20+1].AlarmMsg.EN,
																				'; dec:');																				
AlarmActionArray[log_ID+20*i-20+1].AlarmMsg.EN	:=	CONCAT(AlarmActionArray[log_ID+20*i-20+1].AlarmMsg.EN,
																				LREAL_TO_STRING(GVL_API.stRoolToRool[i].deceleration));
AlarmActionArray[log_ID+20*i-20+1].AlarmMsg.EN	:=	CONCAT(AlarmActionArray[log_ID+20*i-20+1].AlarmMsg.EN,
																				'; rate:');	
AlarmActionArray[log_ID+20*i-20+1].AlarmMsg.EN	:=	CONCAT(AlarmActionArray[log_ID+20*i-20+1].AlarmMsg.EN,
																				DINT_TO_STRING(GVL_API.stRoolToRool[i].rate));	
AlarmActionArray[log_ID+20*i-20+1].AlarmMsg.EN	:=	CONCAT(AlarmActionArray[log_ID+20*i-20+1].AlarmMsg.EN,
																				'; untensionRate:');																						
AlarmActionArray[log_ID+20*i-20+1].AlarmMsg.EN	:=	CONCAT(AlarmActionArray[log_ID+20*i-20+1].AlarmMsg.EN,
																				DINT_TO_STRING(GVL_API.stRoolToRool[i].untension_rate));																					
fbSetAlarm[log_ID+20*i-20+1](
	InUse:=TRUE , 
	EventId:=log_ID+20*i-20+1 , 
	EventActive:=GVL_API.stRoolToRool[i].Initialize, 
	EventClass:=Alm_EventClass.Event , 
	ToTheLogFile:=TRUE, 
	ToTheHistory:=TRUE , 
 );
 
 //SetActivate
AlarmActionArray[log_ID+20*i-20+2].AlarmMsg.EN	:=	CONCAT('Rool-',INT_TO_STRING(i));
AlarmActionArray[log_ID+20*i-20+2].AlarmMsg.EN	:=	CONCAT(AlarmActionArray[log_ID+20*i-20+2].AlarmMsg.EN,
																				' SetActivate');
fbSetAlarm[log_ID+20*i-20+2](
	InUse:=TRUE , 
	EventId:=log_ID+20*i-20+2 , 
	EventActive:=GVL_API.stRoolToRool[i].SetActivate, 
	EventClass:=Alm_EventClass.Event , 
	ToTheLogFile:=TRUE, 
	ToTheHistory:=TRUE , 
 );
 
 //SetReady
AlarmActionArray[log_ID+20*i-20+3].AlarmMsg.EN	:=	CONCAT('Rool-',INT_TO_STRING(i));
AlarmActionArray[log_ID+20*i-20+3].AlarmMsg.EN	:=	CONCAT(AlarmActionArray[log_ID+20*i-20+3].AlarmMsg.EN,
																				' SetReady');
fbSetAlarm[log_ID+20*i-20+3](
	InUse:=TRUE , 
	EventId:=log_ID+20*i-20+3 , 
	EventActive:=GVL_API.stRoolToRool[i].SetReady, 
	EventClass:=Alm_EventClass.Event , 
	ToTheLogFile:=TRUE, 
	ToTheHistory:=TRUE , 
 );
 
 //EnableBrake
AlarmActionArray[log_ID+20*i-20+4].AlarmMsg.EN	:=	CONCAT('Rool-',INT_TO_STRING(i));
AlarmActionArray[log_ID+20*i-20+4].AlarmMsg.EN	:=	CONCAT(AlarmActionArray[log_ID+20*i-20+4].AlarmMsg.EN,
																				' EnableBrake timeout:');
AlarmActionArray[log_ID+20*i-20+4].AlarmMsg.EN	:=	CONCAT(AlarmActionArray[log_ID+20*i-20+4].AlarmMsg.EN,
																				LREAL_TO_STRING(GVL_API.stRoolToRool[i].brake_timeout));																						
																				
fbSetAlarm[log_ID+20*i-20+4](
	InUse:=TRUE , 
	EventId:=log_ID+20*i-20+4 , 
	EventActive:=GVL_API.stRoolToRool[i].EnableBrake, 
	EventClass:=Alm_EventClass.Event , 
	ToTheLogFile:=TRUE, 
	ToTheHistory:=TRUE , 
 );
 
 //DisableBrake
AlarmActionArray[log_ID+20*i-20+5].AlarmMsg.EN	:=	CONCAT('Rool-',INT_TO_STRING(i));
AlarmActionArray[log_ID+20*i-20+5].AlarmMsg.EN	:=	CONCAT(AlarmActionArray[log_ID+20*i-20+5].AlarmMsg.EN,
																				' DisableBrake');																					
																				
fbSetAlarm[log_ID+20*i-20+5](
	InUse:=TRUE , 
	EventId:=log_ID+20*i-20+5 , 
	EventActive:=GVL_API.stRoolToRool[i].DisableBrake, 
	EventClass:=Alm_EventClass.Event , 
	ToTheLogFile:=TRUE, 
	ToTheHistory:=TRUE , 
 ); 
 
 //StartTension
AlarmActionArray[log_ID+20*i-20+6].AlarmMsg.EN	:=	CONCAT('Rool-',INT_TO_STRING(i));
IF GVL_API.stRoolToRool[i].tension_mode THEN 
AlarmActionArray[log_ID+20*i-20+6].AlarmMsg.EN	:=	CONCAT(AlarmActionArray[log_ID+20*i-20+6].AlarmMsg.EN,
																				' inside');
ELSE
AlarmActionArray[log_ID+20*i-20+6].AlarmMsg.EN	:=	CONCAT(AlarmActionArray[log_ID+20*i-20+6].AlarmMsg.EN,
																				' outside');			
END_IF
fbSetAlarm[log_ID+20*i-20+6](
	InUse:=TRUE , 
	EventId:=log_ID+20*i-20+6 , 
	EventActive:=GVL_API.stRoolToRool[i].StartTension, 
	EventClass:=Alm_EventClass.Event , 
	ToTheLogFile:=TRUE, 
	ToTheHistory:=TRUE , 
 ); 
 
 //StopTension
AlarmActionArray[log_ID+20*i-20+7].AlarmMsg.EN	:=	CONCAT('Rool-',INT_TO_STRING(i));
AlarmActionArray[log_ID+20*i-20+7].AlarmMsg.EN	:=	CONCAT(AlarmActionArray[log_ID+20*i-20+7].AlarmMsg.EN,
																				' StopTension timeout:');	
AlarmActionArray[log_ID+20*i-20+7].AlarmMsg.EN	:=	CONCAT(AlarmActionArray[log_ID+20*i-20+7].AlarmMsg.EN,
																				LREAL_TO_STRING(GVL_API.stRoolToRool[i].untension_timeout));	
																				
fbSetAlarm[log_ID+20*i-20+7](
	InUse:=TRUE , 
	EventId:=log_ID+20*i-20+7 , 
	EventActive:=GVL_API.stRoolToRool[i].StopTension, 
	EventClass:=Alm_EventClass.Event , 
	ToTheLogFile:=TRUE, 
	ToTheHistory:=TRUE , 
 ); 					

//	SetOff
AlarmActionArray[log_ID+20*i-20+8].AlarmMsg.EN	:=	CONCAT('Rool-',INT_TO_STRING(i));
AlarmActionArray[log_ID+20*i-20+8].AlarmMsg.EN	:=	CONCAT(AlarmActionArray[log_ID+20*i-20+8].AlarmMsg.EN,
																				' SetOff');	
														
fbSetAlarm[log_ID+20*i-20+8](
	InUse:=TRUE , 
	EventId:=log_ID+20*i-20+8 , 
	EventActive:=GVL_API.stRoolToRool[i].SetOff, 
	EventClass:=Alm_EventClass.Event , 
	ToTheLogFile:=TRUE, 
	ToTheHistory:=TRUE , 
 ); 			 
 
 //ERROR,log_ErrorEnum只能等于一个常数
CASE GVL_API.stRoolToRool[i].error_code OF
0	:	log_ErrorEnum	:=	0	;
1	:	log_ErrorEnum	:=	1	;
2	:	log_ErrorEnum	:=	2	;
3	:	log_ErrorEnum	:=	3	;
4	:	log_ErrorEnum	:=	4	;
5	:	log_ErrorEnum	:=	5	;
6	:	log_ErrorEnum	:=	6	;
7	:	log_ErrorEnum	:=	7	;
8	:	log_ErrorEnum	:=	8	;
666	:	log_ErrorEnum	:=	666	;
 
END_CASE
AlarmActionArray[log_ID+20*i-20+9].AlarmMsg.EN	:=	CONCAT('Rool-',INT_TO_STRING(i));
AlarmActionArray[log_ID+20*i-20+9].AlarmMsg.EN	:=	CONCAT(AlarmActionArray[log_ID+20*i-20+9].AlarmMsg.EN,
																				' Error:');	
AlarmActionArray[log_ID+20*i-20+9].AlarmMsg.EN	:=	CONCAT(AlarmActionArray[log_ID+20*i-20+9].AlarmMsg.EN,
																				TO_STRING(log_ErrorEnum));

fbSetAlarm[log_ID+20*i-20+9](
	InUse:=TRUE , 
	EventId:=log_ID+20*i-20+9 , 
	EventActive:=GVL_API.stRoolToRool[i].error_code<>0 AND GVL_API.stRoolToRool[i].error_code<>666 , 
	EventClass:=Alm_EventClass.Alarm , 
	ToTheLogFile:=TRUE, 
	ToTheHistory:=TRUE , 
 );	
 
//AXIS_ERROR
AlarmActionArray[log_ID+20*i-20+10].AlarmMsg.EN	:=	CONCAT('Rool-',INT_TO_STRING(i));
AlarmActionArray[log_ID+20*i-20+10].AlarmMsg.EN	:=	CONCAT(AlarmActionArray[log_ID+20*i-20+10].AlarmMsg.EN,
																				' Axis_ErrorID:');	
AlarmActionArray[log_ID+20*i-20+10].AlarmMsg.EN	:=CONCAT(AlarmActionArray[log_ID+20*i-20+10].AlarmMsg.EN,
																				UDINT_TO_STRING(FB_RoolToRool[i].REF.Status.ErrorID));
fbSetAlarm[log_ID+20*i-20+10](
	InUse:=TRUE , 
	EventId:=log_ID+20*i-20+10 , 
	EventActive:=FB_RoolToRool[i].REF.Status.Error , 
	EventClass:=Alm_EventClass.Alarm , 
	ToTheLogFile:=TRUE, 
	ToTheHistory:=TRUE , 
 );																						
 END_FOR
 
 //usable
IF GVL_API.stRoolToRool[1].usable THEN 
AlarmActionArray[781].AlarmMsg.EN	:=	'RoolToRool object in a double lane setup ';
ELSE
AlarmActionArray[781].AlarmMsg.EN	:=	'RoolToRool object in a single  lane setup ';
END_IF

ton_old_usable(IN:=NOT ton_old_usable.Q  , PT:=T#200MS , Q=> , ET=> );
IF ton_old_usable.Q THEN 
	old_usable:=GVL_API.stRoolToRool[1].usable ;
END_IF
fbSetAlarm[781](
	InUse:=TRUE , 
	EventId:=781 , 
	EventActive:=old_usable<> GVL_API.stRoolToRool[1].usable, 
	EventClass:=Alm_EventClass.Event , 
	ToTheLogFile:=TRUE, 
	ToTheHistory:=TRUE , 
 );
 
 //isprinting
IF GVL_API.stRoolToRool[1].is_printing THEN 
AlarmActionArray[782].AlarmMsg.EN	:=	'is_printing:TRUE ';
ELSE
AlarmActionArray[782].AlarmMsg.EN	:=	'is_printing:FALSE ';
END_IF

ton_old_isprinting(IN:=NOT ton_old_isprinting.Q  , PT:=T#200MS , Q=> , ET=> );
IF ton_old_isprinting.Q THEN 
	old_isprinting:= GVL_API.stRoolToRool[1].is_printing ;
END_IF
fbSetAlarm[782](
	InUse:=TRUE , 
	EventId:=782 , 
	EventActive:=old_isprinting<> GVL_API.stRoolToRool[1].is_printing, 
	EventClass:=Alm_EventClass.Event , 
	ToTheLogFile:=TRUE, 
	ToTheHistory:=TRUE , 
 );
 
 (*************em-stop*     549*************
AlarmActionArray[783].AlarmMsg.EN	:=	'Rool Error:emergency_error';	

fbSetAlarm[783](
	InUse:=TRUE , 
	EventId:=783 , 
	EventActive:=GVL_API.stRoolToRool[1].error_code=666  , 
	EventClass:=Alm_EventClass.Alarm , 
	ToTheLogFile:=TRUE, 
	ToTheHistory:=TRUE , 
 );	
 *)
END_ACTION

END_PROGRAM

// ---- VISUs/Components/VIS_FootPedal.TcVIS
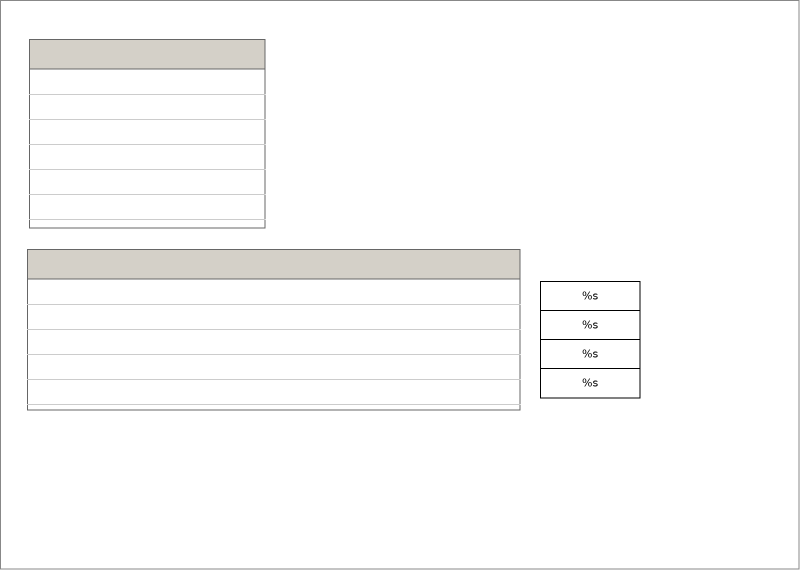
VISUALIZATION VIS_FootPedal  // 800x570
    Table (29,39 236x189), data array: stInput.biFootPedal
        p3854506369: stInput.biFootPedal[INDEX].PedalPressed1
        p1892666644: stInput.biFootPedal[INDEX].PedalPressed2
        p338671338: stInput.biFootPedal[INDEX].PedalPressed3
        Columns.Column.[2].Template: toggle stInput.biFootPedal[INDEX].PedalPressed3
        Columns.Column.[0].Template: toggle stInput.biFootPedal[INDEX].PedalPressed1
        Columns.Column.[1].Template: toggle stInput.biFootPedal[INDEX].PedalPressed2
    Table (27,249 493x161), data array: GVL_API.stFootPedal
        p1218418051: P_FootPedal.FB_FootPedal[INDEX].state
        p746581629: P_FootPedal.FB_FootPedal[INDEX].pressed
        p3104783080: P_FootPedal.FB_FootPedal[INDEX].ton1
        p2501879983: P_FootPedal.FB_FootPedal[INDEX].step
        p7306298: P_FootPedal.FB_FootPedal[INDEX].Reset
        p3854506369: GVL_API.stFootPedal[INDEX].error_code
        p1892666644: GVL_API.stFootPedal[INDEX].state
        p338671338: GVL_API.stFootPedal[INDEX].pressed
        p2170511999: GVL_API.stFootPedal[INDEX].Reset
        p3723444502: GVL_API.stFootPedal[INDEX].debounce_time
        Columns.Column.[4].Template: OnMouseDown: write GVL_API.stFootPedal[INDEX].debounce_time via Default
        Columns.Column.[3].Template: toggle GVL_API.stFootPedal[INDEX].Reset
    Rectangle (540,281 100x30), "%s", text variable: P_FootPedal.FB_FootPedal[1].ton1.ET
    Rectangle (540,310 100x30), "%s", text variable: P_FootPedal.FB_FootPedal[2].ton1.ET
    Rectangle (540,339 100x30), "%s", text variable: P_FootPedal.FB_FootPedal[3].ton1.ET
    Rectangle (540,368 100x30), "%s", text variable: P_FootPedal.FB_FootPedal[4].ton1.ET
END_VISUALIZATION

// ---- VISUs/Components/VIS_Drip_purge.TcVIS
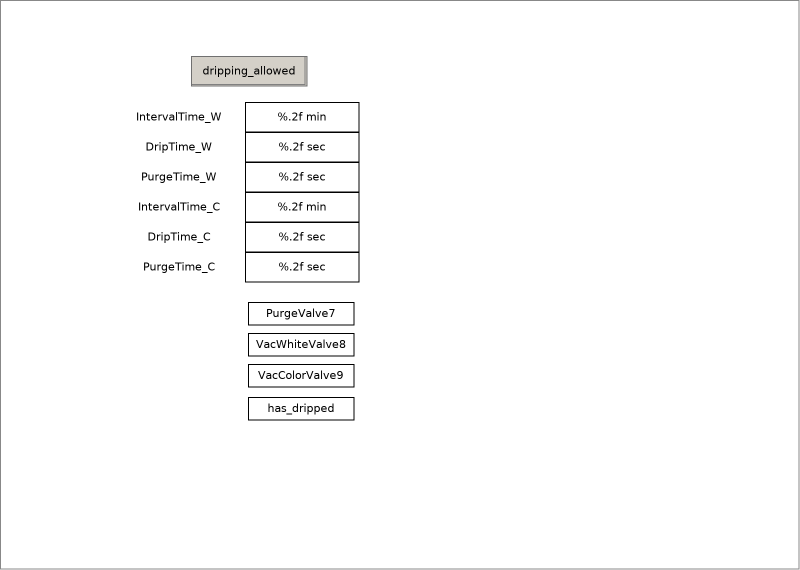
VISUALIZATION VIS_Drip_purge  // 800x570
    Button (191,56 116x30), "dripping_allowed", colour toggle: GVL_API.stMU.dripping_allowed
        toggle GVL_API.stMU.dripping_allowed
    RoundedRectangle (248,302 106x23), "PurgeValve7", colour toggle: P_MaintenanceUnit.FB_drip_purge.PurgeValve7
    Label (122,102 114x30), "IntervalTime_W"
    Label (122,132 114x30), "DripTime_W"
    Label (122,222 114x30), "DripTime_C"
    Label (122,162 114x30), "PurgeTime_W"
    Label (122,192 114x30), "IntervalTime_C"
    Label (122,252 114x30), "PurgeTime_C"
    Rectangle (245,102 114x30), "%.2f min", text variable: GVL_API.stMU.IntervalTime_W
        OnMouseDown: write GVL_API.stMU.IntervalTime_W via Default
    Rectangle (245,132 114x30), "%.2f sec", text variable: GVL_API.stMU.DripTime_W
        OnMouseDown: write GVL_API.stMU.DripTime_W via Default
    Rectangle (245,162 114x30), "%.2f sec", text variable: GVL_API.stMU.PurgeTime_W
        OnMouseDown: write GVL_API.stMU.PurgeTime_W via Default
    Rectangle (245,192 114x30), "%.2f min", text variable: GVL_API.stMU.IntervalTime_C
        OnMouseDown: write GVL_API.stMU.IntervalTime_C via Default
    Rectangle (245,222 114x30), "%.2f sec", text variable: GVL_API.stMU.DripTime_C
        OnMouseDown: write GVL_API.stMU.DripTime_C via Default
    Rectangle (245,252 114x30), "%.2f sec", text variable: GVL_API.stMU.PurgeTime_C
        OnMouseDown: write GVL_API.stMU.PurgeTime_C via Default
    RoundedRectangle (248,333 106x23), "VacWhiteValve8", colour toggle: P_MaintenanceUnit.FB_drip_purge.VacWhiteValve8
    RoundedRectangle (248,364 106x23), "VacColorValve9", colour toggle: P_MaintenanceUnit.FB_drip_purge.VacColorValve9
    RoundedRectangle (248,397 106x23), "has_dripped", colour toggle: GVL_API.stMU.has_dripped
END_VISUALIZATION

// ---- VISUs/Components/VIS_SystemEnvironment.TcVIS
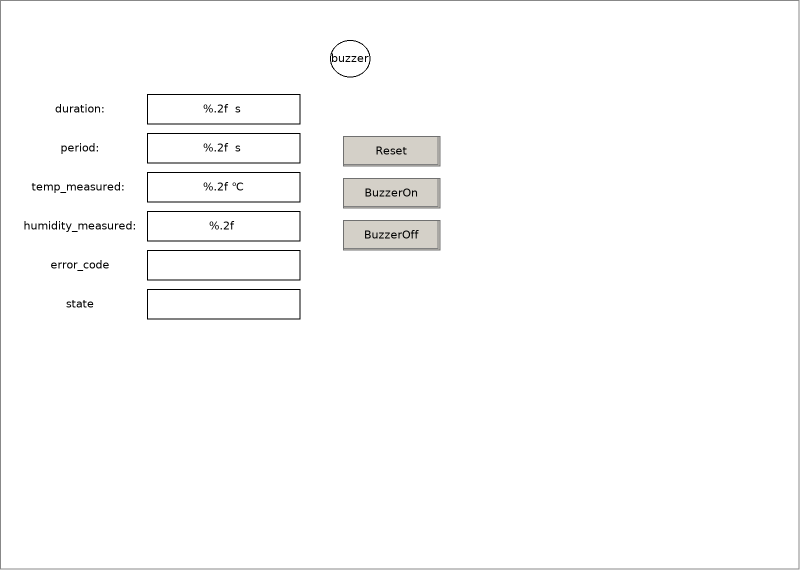
VISUALIZATION VIS_SystemEnvironment  // 800x570
    Button (343,178 97x30), "BuzzerOn", colour toggle: GVL_API.stSystemEnvironment.BuzzerOn
        toggle GVL_API.stSystemEnvironment.BuzzerOn
    Button (343,136 97x30), "Reset", colour toggle: GVL_API.stSystemEnvironment.Reset
        toggle GVL_API.stSystemEnvironment.Reset
    Button (343,220 97x30), "BuzzerOff", colour toggle: GVL_API.stSystemEnvironment.BuzzerOff
        toggle GVL_API.stSystemEnvironment.BuzzerOff
    Ellipse (330,40 40x37), "buzzer", colour toggle: stOutput.bqBuzzer
    Rectangle (147,94 153x30), "%.2f s", text variable: GVL_API.stSystemEnvironment.duration
        OnMouseDown: write GVL_API.stSystemEnvironment.duration via Default
    Rectangle (147,133 153x30), "%.2f s", text variable: GVL_API.stSystemEnvironment.period
        OnMouseDown: write GVL_API.stSystemEnvironment.period via Default
    Rectangle (147,211 153x30), "%.2f", text variable: GVL_API.stSystemEnvironment.humidity_measured
        OnMouseDown: write GVL_API.stRoolToRool[1].acceleration via Default
    Rectangle (147,172 153x30), "%.2f ℃", text variable: GVL_API.stSystemEnvironment.temp_measured
    Rectangle (147,250 153x30), text list: 'TextList_EnvironmentError', text index: GVL_API.stSystemEnvironment.error_code
    Rectangle (147,289 153x30), text list: 'TextList_EnvironmentState', text index: GVL_API.stSystemEnvironment.state
    Label (15,250 130x30), "error_code"
    Label (15,289 130x30), "state"
    Label (15,211 130x30), "humidity_measured:"
    Label (15,172 130x30), "temp_measured:"
    Label (15,133 130x30), "period:"
    Label (15,94 130x30), "duration:"
END_VISUALIZATION

// ---- VISUs/Components/VIS_ISS.TcVIS
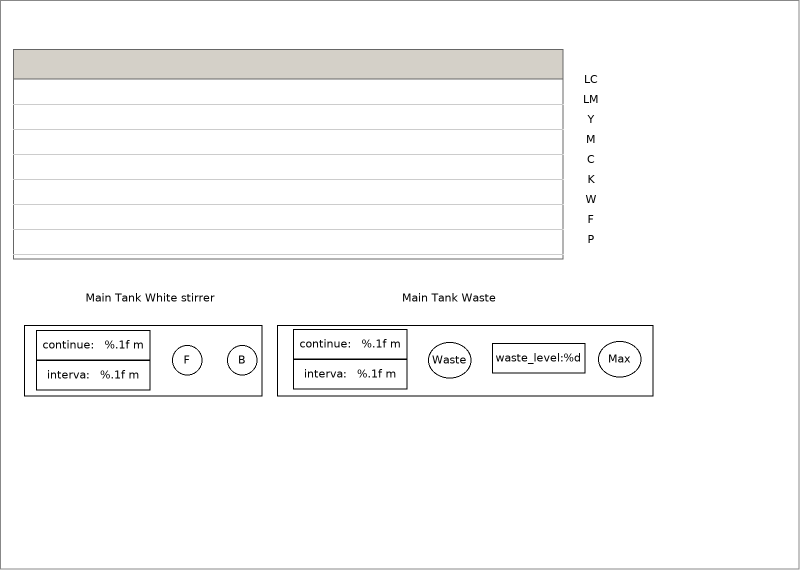
VISUALIZATION VIS_ISS  // 800x570
    RoundedRectangle (277,325 376x71)
    RoundedRectangle (24,325 238x71)
    Table (13,49 550x210), data array: GVL_API.stISS
        p3854506369: GVL_API.stISS[INDEX].error_code
        p1892666644: GVL_API.stISS[INDEX].state
        p338671338: GVL_API.stISS[INDEX].mainTankLevel
        p2170511999: GVL_API.stISS[INDEX].Init_Done
        p3723444502: GVL_API.stISS[INDEX].Error
        p1218418051: GVL_API.stISS[INDEX].Initialize
        p746581629: GVL_API.stISS[INDEX].Setoff
        p3104783080: GVL_API.stISS[INDEX].sensor_blink
        Columns.Column.[5].Template: toggle GVL_API.stISS[INDEX].Initialize
        Columns.Column.[6].Template: toggle GVL_API.stISS[INDEX].Setoff
    Rectangle (36,330 114x30), "continue: %.1f m", text variable: HMI_SetStirrer_continueTime
        OnMouseDown: write HMI_SetStirrer_continueTime via Default, min 0.01
    Rectangle (36,360 114x30), "interva: %.1f m", text variable: HMI_SetStirrer_intervalTime
        OnMouseDown: write HMI_SetStirrer_intervalTime via Default, min 0.5
    Ellipse (172,345 30x30), "F", colour toggle: stOutput.bqStirrerWorkingF
    Ellipse (227,345 30x30), "B", colour toggle: stOutput.bqStirrerWorkingB
    Ellipse (428,342 43x36), "Waste", colour toggle: stOutput.bqWastePump
    Rectangle (293,329 114x30), "continue: %.1f m", text variable: HMI_SetWaste_continueTime
        OnMouseDown: write HMI_SetWaste_continueTime via Default
    Rectangle (293,359 114x30), "interva: %.1f m", text variable: HMI_SetWaste_intervalTime
        OnMouseDown: write HMI_SetWaste_intervalTime via Default, min 0.1
    Rectangle (492,343 93x30), "waste_level:%d", text variable: GVL.MainTankLevel[10]
    Ellipse (598,341 43x36), "Max", colour toggle: GVL_API.stMU.waste_maximum_level
    Label (567,72 48x15), "LC"
    Label (567,92 48x15), "LM"
    Label (567,112 48x15), "Y"
    Label (567,132 48x15), "M"
    Label (567,152 48x15), "C"
    Label (567,192 48x15), "W"
    Label (567,232 48x15), "P"
    Label (567,172 48x15), "K"
    Label (567,212 48x15), "F"
    Label (68,283 164x30), "Main Tank White stirrer"
    Label (367,283 164x30), "Main Tank Waste"
END_VISUALIZATION

// ---- VISUs/Components/VIS_MU.TcVIS
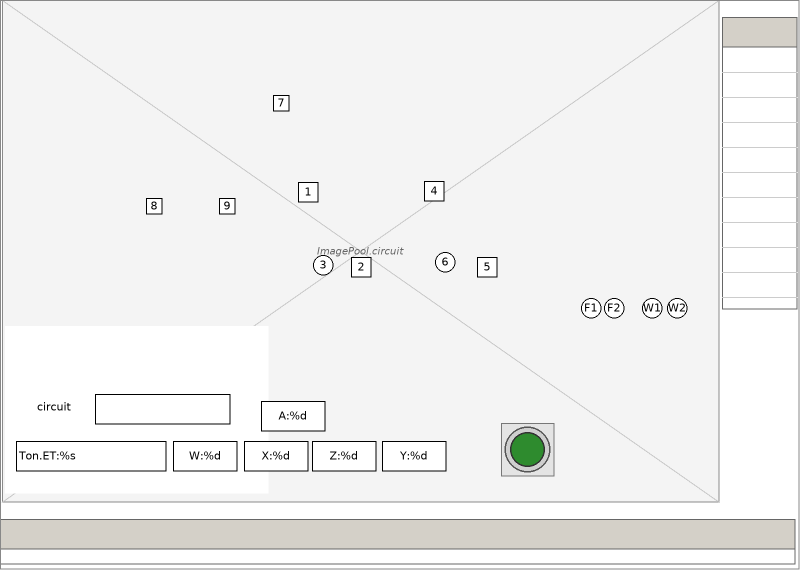
VISUALIZATION VIS_MU  // 800x570
    Image (2,0 717x502), image: ImagePool.circuit
    Ellipse (313,255 20x20), "3", colour toggle: stOutput.bqSubCircPumpWorking[1]
    Rectangle (351,257 20x20), "2", colour toggle: GVL.inklevel_W_L_BOT
        toggle stInput.biSubInkTankLevel[15]
    Ellipse (435,252 20x20), "6", colour toggle: stOutput.bqSubCircPumpWorking[2]
    Rectangle (477,257 20x20), "5", colour toggle: GVL.inklevel_W_R_BOT
        toggle stInput.biSubInkTankLevel[18]
    Rectangle (298,182 20x20), "1", colour toggle: GVL.inklevel_W_L_TOP
        toggle stInput.biSubInkTankLevel[16]
    Rectangle (424,181 20x20), "4", colour toggle: GVL.inklevel_W_R_TOP
        toggle stInput.biSubInkTankLevel[17]
    Rectangle (146,198 16x16), "8", colour toggle: stOutput.bqVacValve_W
    Rectangle (219,198 16x16), "9", colour toggle: stOutput.bqVacValve_C
    Rectangle (273,95 16x16), "7", colour toggle: stOutput.bqPurValve
    Ellipse (581,298 20x20), "F1", colour toggle: stOutput.bqFillPumpWorking[19]
    Ellipse (604,298 20x20), "F2", colour toggle: stOutput.bqFillPumpWorking[20]
    Ellipse (642,298 20x20), "W1", colour toggle: stOutput.bqFillPumpWorking[13]
    Ellipse (667,298 20x20), "W2", colour toggle: stOutput.bqFillPumpWorking[15]
    Rectangle (5,326 263x167)
    Table (0,519 795x45), data array: P_MaintenanceUnit.FB_Auto_Cycles_Swap
        p3854506369: P_MaintenanceUnit.FB_Auto_Cycles_Swap.Sensor1
        p1892666644: P_MaintenanceUnit.FB_Auto_Cycles_Swap.Sensor4
        p338671338: P_MaintenanceUnit.FB_Auto_Cycles_Swap.Circ_Pump_L
        p2170511999: P_MaintenanceUnit.FB_Auto_Cycles_Swap.Circ_Pump_R
        p3723444502: P_MaintenanceUnit.FB_Auto_Cycles_Swap.Circ_normal_error
        p1218418051: P_MaintenanceUnit.FB_Auto_Cycles_Swap.btPurge
        p746581629: P_MaintenanceUnit.FB_Auto_Cycles_Swap.state
        p3104783080: P_MaintenanceUnit.FB_Auto_Cycles_Swap.error_code
        p2501879983: P_MaintenanceUnit.FB_Auto_Cycles_Swap.SwapInfo
        p7306298: P_MaintenanceUnit.FB_Auto_Cycles_Swap.VacValve_V8
        p1933151965: P_MaintenanceUnit.FB_Auto_Cycles_Swap.PurValve_V7
        p3863566920: P_MaintenanceUnit.FB_Auto_Cycles_Swap.alternate_Pumping
        p2192122294: P_MaintenanceUnit.FB_Auto_Cycles_Swap.Swapping_Done
        p400160035: P_MaintenanceUnit.FB_Auto_Cycles_Swap.Error
        p1265227338: P_MaintenanceUnit.FB_Auto_Cycles_Swap.step
        p3726181087: P_MaintenanceUnit.FB_Auto_Cycles_Swap.stepA
        p3136911649: P_MaintenanceUnit.FB_Auto_Cycles_Swap.stepB1
        p797552052: P_MaintenanceUnit.FB_Auto_Cycles_Swap.stepB2
        p60375027: P_MaintenanceUnit.FB_Auto_Cycles_Swap.Ton
        p2531912550: P_MaintenanceUnit.FB_Auto_Cycles_Swap.ton7
        p693678525: P_MaintenanceUnit.FB_Auto_Cycles_Swap.ton10
        p3156763944: P_MaintenanceUnit.FB_Auto_Cycles_Swap.FB_SQUARE
        p3636993750: P_MaintenanceUnit.FB_Auto_Cycles_Swap.W
        p1303956035: P_MaintenanceUnit.FB_Auto_Cycles_Swap.X
        p285796650: P_MaintenanceUnit.FB_Auto_Cycles_Swap.A
        p2222472639: P_MaintenanceUnit.FB_Auto_Cycles_Swap.Z
        p3768075841: P_MaintenanceUnit.FB_Auto_Cycles_Swap.Y
        p1978176212: P_MaintenanceUnit.FB_Auto_Cycles_Swap.cycle_r_trig1
        p1509425299: P_MaintenanceUnit.FB_Auto_Cycles_Swap.cycle_r_trig2
        p3431519238: P_MaintenanceUnit.FB_Auto_Cycles_Swap.cycle_x1
        p2846402210: P_MaintenanceUnit.FB_Auto_Cycles_Swap.cycle_x2
        p1020817975: P_MaintenanceUnit.FB_Auto_Cycles_Swap.purge_F_trig
        p1480067529: P_MaintenanceUnit.FB_Auto_Cycles_Swap.dely_off_setoff
        p3444104540: P_MaintenanceUnit.FB_Auto_Cycles_Swap.dely_emstop
        p76032672: GVL_API.stMU.Initialize
        p1617449310: GVL_API.stMU.Swap
        p4112025035: P_MaintenanceUnit.FB_Auto_Cycles_Swap.CYCLE
        p3641186188: GVL_API.stMU.SetOff
        p633067465: initialize
        p1398730484: swap
        p3327948760: P_MaintenanceUnit.FB_Auto_Cycles_Swap.initialize
        p1777678866: P_MaintenanceUnit.FB_Auto_Cycles_Swap.swap
        p1879929205: P_MaintenanceUnit.FB_Auto_Cycles_Swap.setoff
        Columns.Column.[37].Template: OnMouseDown: write P_MaintenanceUnit.FB_Auto_Cycles_Swap.CYCLE via Default, min 0, max 1
        Columns.Column.[38].Template: toggle GVL_API.stMU.SetOff
        Columns.Column.[35].Template: toggle GVL_API.stMU.Initialize
        Columns.Column.[36].Template: toggle GVL_API.stMU.Swap
    Rectangle (16,441 150x30), "Ton.ET:%s", text variable: P_MaintenanceUnit.FB_Auto_Cycles_Swap.Ton.ET
    Table (722,17 75x292), data array: T
        p3854506369: T[INDEX]
        Columns.Column.[0].Template: OnMouseDown: write T[INDEX] via Default
    Rectangle (173,441 64x30), "W:%d", text variable: P_MaintenanceUnit.FB_Auto_Cycles_Swap.W
    Rectangle (244,441 64x30), "X:%d", text variable: P_MaintenanceUnit.FB_Auto_Cycles_Swap.X
    PushSwitch (500,423 55x53), variable: stInput.btPurge, behaviour: TAP, style: Switch-PushSwitch-Green
    Rectangle (312,441 64x30), "Z:%d", text variable: P_MaintenanceUnit.FB_Auto_Cycles_Swap.Z
    Rectangle (382,441 64x30), "Y:%d", text variable: P_MaintenanceUnit.FB_Auto_Cycles_Swap.Y
    Rectangle (95,394 135x30), text list: 'TextList_SubTank_circuit', text index: SubTankInk_type
        OnMouseDown: write HMI_CircPump1_V via Default, min 0, max 5
    Label (24,392 60x30), "circuit"
    Rectangle (261,401 64x30), "A:%d", text variable: P_MaintenanceUnit.FB_Auto_Cycles_Swap.A
END_VISUALIZATION

// ---- VISUs/Components/VIS_RTR_1.TcVIS
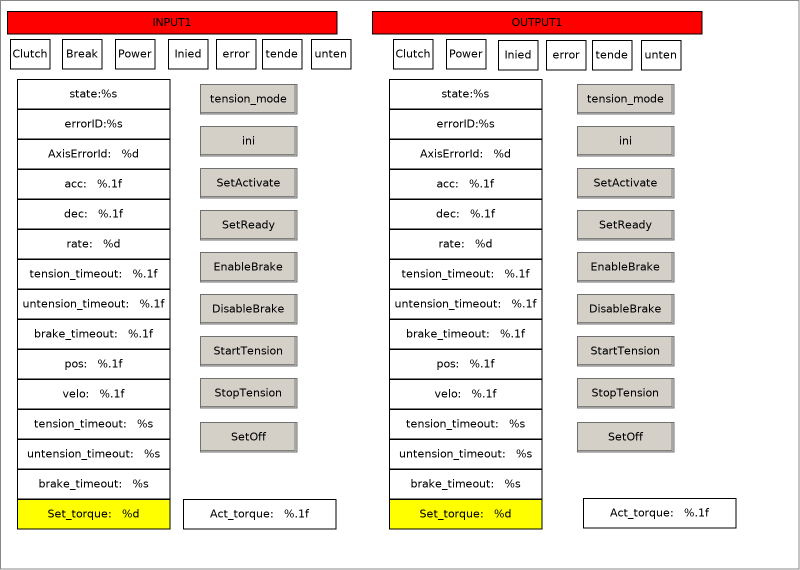
VISUALIZATION VIS_RTR_1  // 800x570
    RoundedRectangle (372,11 330x23), "OUTPUT1"
    RoundedRectangle (7,11 330x23), "INPUT1"
    Button (200,126 97x30), "ini", colour toggle: GVL_API.stRoolToRool[1].Initialize
        toggle GVL_API.stRoolToRool[1].Initialize
    Button (200,84 97x30), "tension_mode", colour toggle: GVL_API.stRoolToRool[1].tension_mode
        toggle GVL_API.stRoolToRool[1].tension_mode
    Button (200,168 97x30), "SetActivate", colour toggle: GVL_API.stRoolToRool[1].SetActivate
        toggle GVL_API.stRoolToRool[1].SetActivate
    Button (200,294 97x30), "DisableBrake", colour toggle: GVL_API.stRoolToRool[1].DisableBrake
        toggle GVL_API.stRoolToRool[1].DisableBrake
    Button (200,210 97x30), "SetReady", colour toggle: GVL_API.stRoolToRool[1].SetReady
        toggle GVL_API.stRoolToRool[1].SetReady
    Button (200,252 97x30), "EnableBrake", colour toggle: GVL_API.stRoolToRool[1].EnableBrake
        toggle GVL_API.stRoolToRool[1].EnableBrake
    Button (200,336 97x30), "StartTension", colour toggle: GVL_API.stRoolToRool[1].StartTension
        toggle GVL_API.stRoolToRool[1].StartTension
    Button (200,378 97x30), "StopTension", colour toggle: GVL_API.stRoolToRool[1].StopTension
        toggle GVL_API.stRoolToRool[1].StopTension
    Button (200,422 97x30), "SetOff", colour toggle: GVL_API.stRoolToRool[1].SetOff
        toggle GVL_API.stRoolToRool[1].SetOff
    RoundedRectangle (62,39 40x30), "Break", colour toggle: stOutput.bqBreakPower[1]
    RoundedRectangle (10,39 40x30), "Clutch", colour toggle: stOutput .bqCluthOut[1]
    Rectangle (17,79 153x30), "state:%s", colour toggle: GVL_API.stRoolToRool[1].state=100, text list: 'TextList_RTRstate', text index: GVL_API.stRoolToRool[1].state
    Rectangle (17,109 153x30), "errorID:%s", colour toggle: GVL_API.stRoolToRool[1].error_code<>0, text list: 'TextList_RTR_errorid', text index: GVL_API.stRoolToRool[1].error_code
    Rectangle (17,169 153x30), "acc: %.1f", text variable: GVL_API.stRoolToRool[1].acceleration
        OnMouseDown: write GVL_API.stRoolToRool[1].acceleration via Default
    Rectangle (17,199 153x30), "dec: %.1f", text variable: GVL_API.stRoolToRool[1].deceleration
        OnMouseDown: write GVL_API.stRoolToRool[1].deceleration via Default
    Rectangle (17,229 153x30), "rate: %d", text variable: GVL_API.stRoolToRool[1].rate
        OnMouseDown: write GVL_API.stRoolToRool[1].rate via Default
    Rectangle (17,259 153x30), "tension_timeout: %.1f", text variable: GVL_API.stRoolToRool[1].tension_timeout
        OnMouseDown: write GVL_API.stRoolToRool[1].tension_timeout via Default
    Rectangle (17,289 153x30), "untension_timeout: %.1f", text variable: GVL_API.stRoolToRool[1].untension_timeout
        OnMouseDown: write GVL_API.stRoolToRool[1].untension_timeout via Default
    Rectangle (17,319 153x30), "brake_timeout: %.1f", text variable: GVL_API.stRoolToRool[1].brake_timeout
        OnMouseDown: write GVL_API.stRoolToRool[1].brake_timeout via Default
    Rectangle (17,139 153x30), "AxisErrorId: %d", text variable: GVL_API.stRoolToRool[1].AxisErrorId
    Rectangle (389,79 153x30), "state:%s", colour toggle: GVL_API.stRoolToRool[2].state=100, text list: 'TextList_RTRstate', text index: GVL_API.stRoolToRool[2].state
    Rectangle (389,109 153x30), "errorID:%s", colour toggle: GVL_API.stRoolToRool[2].error_code<>0, text list: 'TextList_RTR_errorid', text index: GVL_API.stRoolToRool[2].error_code
    Rectangle (389,169 153x30), "acc: %.1f", text variable: GVL_API.stRoolToRool[2].acceleration
        OnMouseDown: write GVL_API.stRoolToRool[2].acceleration via Default
    Rectangle (389,199 153x30), "dec: %.1f", text variable: GVL_API.stRoolToRool[2].deceleration
        OnMouseDown: write GVL_API.stRoolToRool[2].deceleration via Default
    Rectangle (389,229 153x30), "rate: %d", text variable: GVL_API.stRoolToRool[2].rate
        OnMouseDown: write GVL_API.stRoolToRool[2].rate via Default
    Rectangle (389,259 153x30), "tension_timeout: %.1f", text variable: GVL_API.stRoolToRool[2].tension_timeout
        OnMouseDown: write GVL_API.stRoolToRool[2].tension_timeout via Default
    Rectangle (389,289 153x30), "untension_timeout: %.1f", text variable: GVL_API.stRoolToRool[2].untension_timeout
        OnMouseDown: write GVL_API.stRoolToRool[2].untension_timeout via Default
    Rectangle (389,319 153x30), "brake_timeout: %.1f", text variable: GVL_API.stRoolToRool[2].brake_timeout
        OnMouseDown: write GVL_API.stRoolToRool[2].brake_timeout via Default
    Rectangle (389,139 153x30), "AxisErrorId: %d", text variable: GVL_API.stRoolToRool[2].AxisErrorId
    RoundedRectangle (393,39 40x30), "Clutch", colour toggle: stOutput .bqCluthOut[2]
    Button (577,126 97x30), "ini", colour toggle: GVL_API.stRoolToRool[2].Initialize
        toggle GVL_API.stRoolToRool[2].Initialize
    Button (577,84 97x30), "tension_mode", colour toggle: GVL_API.stRoolToRool[2].tension_mode
        toggle GVL_API.stRoolToRool[2].tension_mode
    Button (577,168 97x30), "SetActivate", colour toggle: GVL_API.stRoolToRool[2].SetActivate
        toggle GVL_API.stRoolToRool[2].SetActivate
    Button (577,294 97x30), "DisableBrake", colour toggle: GVL_API.stRoolToRool[2].DisableBrake
        toggle GVL_API.stRoolToRool[1].DisableBrake
    Button (577,210 97x30), "SetReady", colour toggle: GVL_API.stRoolToRool[2].SetReady
        toggle GVL_API.stRoolToRool[2].SetReady
    Button (577,252 97x30), "EnableBrake", colour toggle: GVL_API.stRoolToRool[2].EnableBrake
        toggle GVL_API.stRoolToRool[2].EnableBrake
    Button (577,336 97x30), "StartTension", colour toggle: GVL_API.stRoolToRool[2].StartTension
        toggle GVL_API.stRoolToRool[2].StartTension
    Button (577,378 97x30), "StopTension", colour toggle: GVL_API.stRoolToRool[2].StopTension
        toggle GVL_API.stRoolToRool[2].StopTension
    Button (577,422 97x30), "SetOff", colour toggle: GVL_API.stRoolToRool[2].SetOff
        toggle GVL_API.stRoolToRool[2].SetOff
    RoundedRectangle (115,39 40x30), "Power", colour toggle: P_RollToRoll.FB_RoolToRool[1].REF.Status.ControlLoopClosed
    RoundedRectangle (446,39 40x30), "Power", colour toggle: P_RollToRoll.FB_RoolToRool[2].REF.Status.ControlLoopClosed
    Rectangle (17,349 153x30), "pos: %.1f", text variable: P_RollToRoll.FB_RoolToRool[1].REF.NcToPlc.ActPos
        OnMouseDown: write GVL_API.stRoolToRool[1].brake_timeout via Default
    Rectangle (17,379 153x30), "velo: %.1f", text variable: P_RollToRoll.FB_RoolToRool[1].REF.NcToPlc.ActVelo
        OnMouseDown: write GVL_API.stRoolToRool[1].brake_timeout via Default
    Rectangle (389,349 153x30), "pos: %.1f", text variable: P_RollToRoll.FB_RoolToRool[2].REF.NcToPlc.ActPos
        OnMouseDown: write GVL_API.stRoolToRool[1].brake_timeout via Default
    Rectangle (389,379 153x30), "velo: %.1f", text variable: P_RollToRoll.FB_RoolToRool[2].REF.NcToPlc.ActVelo
        OnMouseDown: write GVL_API.stRoolToRool[1].brake_timeout via Default
    Rectangle (17,409 153x30), "tension_timeout: %s", text variable: P_RollToRoll.FB_RoolToRool[1].tension_ton.ET
    Rectangle (17,439 153x30), "untension_timeout: %s", text variable: P_RollToRoll.FB_RoolToRool[1].untension_ton.ET
    Rectangle (17,469 153x30), "brake_timeout: %s", text variable: P_RollToRoll.FB_RoolToRool[1].enbreak_ton.ET
    Rectangle (389,409 153x30), "tension_timeout: %s", text variable: P_RollToRoll.FB_RoolToRool[2].tension_ton.ET
    Rectangle (389,439 153x30), "untension_timeout: %s", text variable: P_RollToRoll.FB_RoolToRool[2].untension_ton.ET
    Rectangle (389,469 153x30), "brake_timeout: %s", text variable: P_RollToRoll.FB_RoolToRool[2].enbreak_ton.ET
    Rectangle (17,499 153x30), "Set_torque: %d", text variable: HMI_RTR_set_Torque[1]
        OnMouseDown: write HMI_RTR_set_Torque[1] via Default, min 0, max 100
    Rectangle (389,499 153x30), "Set_torque: %d", text variable: HMI_RTR_set_Torque[2]
        OnMouseDown: write HMI_RTR_set_Torque[2] via Default, min 0, max 100
    Rectangle (183,499 153x30), "Act_torque: %.1f", text variable: P_RollToRoll.FB_RoolToRool[1].REF.NcToPlc.ActTorque
    Rectangle (583,498 153x30), "Act_torque: %.1f", text variable: P_RollToRoll.FB_RoolToRool[2].REF.NcToPlc.ActTorque
    RoundedRectangle (168,39 40x30), "Inied", colour toggle: P_RollToRoll.FB_RoolToRool[1].Initialized
    RoundedRectangle (216,39 40x30), "error", colour toggle: P_RollToRoll.FB_RoolToRool[1].error
    RoundedRectangle (262,39 40x30), "tende", colour toggle: P_RollToRoll.FB_RoolToRool[1].tensioned
    RoundedRectangle (311,39 40x30), "unten", colour toggle: P_RollToRoll.FB_RoolToRool[1].untensioned
    RoundedRectangle (498,40 40x30), "Inied", colour toggle: P_RollToRoll.FB_RoolToRool[2].Initialized
    RoundedRectangle (546,40 40x30), "error", colour toggle: P_RollToRoll.FB_RoolToRool[2].error
    RoundedRectangle (592,40 40x30), "tende", colour toggle: P_RollToRoll.FB_RoolToRool[2].tensioned
    RoundedRectangle (641,40 40x30), "unten", colour toggle: P_RollToRoll.FB_RoolToRool[2].untensioned
END_VISUALIZATION

// ---- VISUs/Components/VIS_SaftyGuard.TcVIS
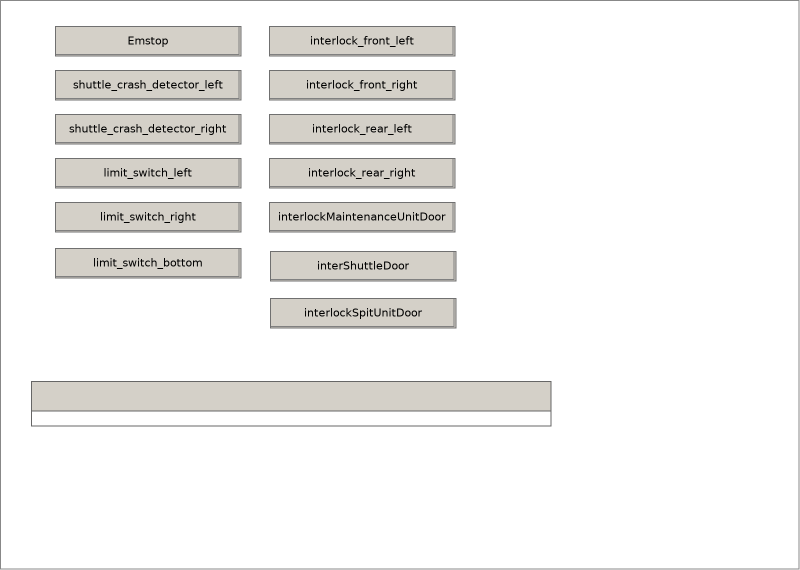
VISUALIZATION VIS_SaftyGuard  // 800x570
    Button (55,26 186x30), "Emstop", colour toggle: GVL_API.stSafetyGuard.emergency_stop
    Button (55,70 186x30), "shuttle_crash_detector_left", colour toggle: GVL_API.stSafetyGuard.shuttle_crash_detector_left
    Button (55,114 186x30), "shuttle_crash_detector_right", colour toggle: GVL_API.stSafetyGuard.shuttle_crash_detector_right
    Button (55,158 186x30), "limit_switch_left", colour toggle: GVL_API.stSafetyGuard.limit_switch_left
    Button (55,202 186x30), "limit_switch_right", colour toggle: GVL_API.stSafetyGuard.limit_switch_right
    Button (269,26 186x30), "interlock_front_left", colour toggle: GVL_API.stSafetyGuard.interlock_front_left
    Button (269,70 186x30), "interlock_front_right", colour toggle: GVL_API.stSafetyGuard.interlock_front_right
    Button (269,114 186x30), "interlock_rear_left", colour toggle: GVL_API.stSafetyGuard.interlock_rear_left
    Button (269,158 186x30), "interlock_rear_right", colour toggle: GVL_API.stSafetyGuard.interlock_rear_right
    Button (269,202 186x30), "interlockMaintenanceUnitDoor", colour toggle: GVL_API.stSafetyGuard.Interlock_maintenace_door, pressed state: P_TwinSAFE.biinterlock[5]
    Button (270,298 186x30), "interlockSpitUnitDoor", colour toggle: GVL_API.stSafetyGuard.Interlock_spit_door
    Button (270,251 186x30), "interShuttleDoor", colour toggle: GVL_API.stSafetyGuard.interlock_shuttle_door
    Button (55,248 186x30), "limit_switch_bottom", colour toggle: GVL_API.stSafetyGuard.limit_switch_bottom
    Table (31,381 520x45), data array: P_SafetyGuard.FB_SafetyGuard
        p3854506369: P_SafetyGuard.FB_SafetyGuard.shuttle_crash_detector
        p1892666644: P_SafetyGuard.FB_SafetyGuard.emergency_stop
        p338671338: P_SafetyGuard.FB_SafetyGuard.limit_switch
        p2170511999: P_SafetyGuard.FB_SafetyGuard.interlock_triggered
        p3723444502: P_SafetyGuard.FB_SafetyGuard.LightCurtainTriggered
        p1218418051: P_SafetyGuard.FB_SafetyGuard.error_code
        p746581629: P_SafetyGuard.FB_SafetyGuard.state
        p3104783080: P_SafetyGuard.FB_SafetyGuard.step
        p2501879983: GVL_API.stSafetyGuard.Initialize
        p7306298: GVL_API.stSafetyGuard.SetOff
        p1037165547: P_SafetyGuard.FB_SafetyGuard.Initialize
        p1488378029: P_SafetyGuard.FB_SafetyGuard.SetOff
        Columns.Column.[5].Template: P_SafetyGuard.FB_SafetyGuard.error_code<>0
        Columns.Column.[8].Template: toggle GVL_API.stSafetyGuard.Initialize
        Columns.Column.[9].Template: toggle GVL_API.stSafetyGuard.SetOff
END_VISUALIZATION

// ---- VISUs/HMI_IO监控文字/EL1809_S_2.TcTLO
TEXTLIST EL1809_S_2
  1 = 'SubInkTankLevel P2' | chinese: '二级墨盒液位图层2' | Chinese: '二级墨盒液位图层2'
  2 = 'SubInkTankLevel W1' | chinese: '二级墨盒液位W1' | Chinese: '二级墨盒液位W1'
  3 = 'SubInkTankLevel W2' | chinese: '二级墨盒液位W2' | Chinese: '二级墨盒液位W2'
  4 = 'SubInkTankLevel W3' | chinese: '二级墨盒液位W3' | Chinese: '二级墨盒液位W3'
  5 = 'SubInkTankLevel W4' | chinese: '二级墨盒液位W4' | Chinese: '二级墨盒液位W4'
  6 = 'ProtectTankLevel_C' | chinese: '真空保护瓶液位1' | Chinese: '真空保护瓶液位1'
  7 = 'ProtectTankLevel_W' | chinese: '真空保护瓶液位2' | Chinese: '真空保护瓶液位2'
  8 = 'Purge button' | chinese: '正压按钮' | Chinese: '正压按钮'
  9 = 'Color vac button' | chinese: '彩色正负压切换按钮' | Chinese: '彩色正负压切换按钮'
  10 = 'White vac button' | chinese: '白色正负压切换按钮' | Chinese: '白色正负压切换按钮'
  11 = ''
  12 = ''
  13 = ''
  14 = ''
  15 = ''
  16 = ''
   = ''
END_TEXTLIST

// ---- VISUs/HMI_IO监控文字/EL1904_M_3.TcTLO
TEXTLIST EL1904_M_3
  1 = 'interlock_out_cover' | chinese: 'OUT_透明盖' | Chinese: 'OUT_透明盖'
  2 = 'interlock_out_cover' | chinese: 'OUT_透明盖' | Chinese: 'OUT_透明盖'
  3 = 'interlock_out_left_door' | chinese: 'OUT_左侧上下门' | Chinese: 'OUT_左侧上下门'
  4 = 'interlock_out_left_door' | chinese: 'OUT_左侧上下门' | Chinese: 'OUT_左侧上下门'
   = ''
END_TEXTLIST

// ---- VISUs/HMI_IO监控文字/EL1904_M_4.TcTLO
TEXTLIST EL1904_M_4
  1 = 'interlock_out_right_door' | chinese: 'OUT_右侧门' | Chinese: 'OUT_右侧门'
  2 = 'interlock_out_right_door' | chinese: 'OUT_右侧门' | Chinese: 'OUT_右侧门'
  3 = 'Reset' | chinese: '复位' | Chinese: '复位'
  4 = ''
   = ''
END_TEXTLIST

// ---- VISUs/HMI_IO监控文字/EL1904_M_5.TcTLO
TEXTLIST EL1904_M_5
  1 = 'Safety output feedback 1' | chinese: '安全输出反馈1' | Chinese: '安全输出反馈1'
  2 = 'Safety output feedback 2' | chinese: '安全输出反馈2' | Chinese: '安全输出反馈2'
  3 = 'Safety output feedback 3' | chinese: '安全输出反馈3' | Chinese: '安全输出反馈3'
  4 = 'Safety output feedback 4' | chinese: '安全输出反馈4' | Chinese: '安全输出反馈4'
   = ''
END_TEXTLIST

// ---- VISUs/HMI_IO监控文字/EL2809_M_1.TcTLO
TEXTLIST EL2809_M_1
  1 = 'F Pump1' | chinese: '清洗液泵1' | Chinese: '图层泵1'
  2 = 'F Pump2' | chinese: '清洗液泵2' | Chinese: '图层泵2'
  3 = 'W ink tank stirring_F' | chinese: '白墨瓶搅拌（正转）' | Chinese: '白墨瓶搅拌（正转）'
  4 = 'W ink tank stirring_B' | chinese: '白墨瓶搅拌（反转）' | Chinese: '白墨瓶搅拌（反转）'
  5 = 'LED_C' | chinese: '墨瓶C  LED' | Chinese: '墨瓶C  LED'
  6 = 'LED_Y' | chinese: '墨瓶Y  LED' | Chinese: '墨瓶Y  LED'
  7 = 'LED_M' | chinese: '墨瓶M  LED' | Chinese: '墨瓶M  LED'
  8 = 'LED_K' | chinese: '墨瓶K  LED' | Chinese: '墨瓶K  LED'
  9 = 'LED_LC' | chinese: '墨瓶LC  LED' | Chinese: '墨瓶LC  LED'
  10 = 'LED_LM' | chinese: '墨瓶LM  LED' | Chinese: '墨瓶LM  LED'
  11 = 'LED_P' | chinese: '墨瓶P LED' | Chinese: '墨瓶W  LED'
  12 = 'LED_W' | chinese: '墨瓶W LED' | Chinese: '墨瓶清洗液  LED'
  13 = 'LED_F' | chinese: '墨瓶F  LED' | Chinese: '墨瓶图层  LED'
  14 = 'LED_Waste' | chinese: '墨瓶废液  LED' | Chinese: '墨瓶废液  LED'
  15 = 'Waste liquid  fan' | chinese: '废液吸风扇' | Chinese: '废液吸风扇'
  16 = 'Waste Pump' | chinese: '废液泵' | Chinese: '废液泵'
   = ''
END_TEXTLIST

// ---- VISUs/HMI_IO监控文字/EL2809_M_2.TcTLO
TEXTLIST EL2809_M_2
  1 = 'Unwinding L Brake' | chinese: '放卷L_刹车' | Chinese: '放卷L_刹车'
  2 = 'Un_L Clutch Out' | chinese: '放卷L_离合器out' | Chinese: '放卷L_离合器out'
  3 = 'Un_L Clutch RST' | chinese: '放卷L_离合器rst' | Chinese: '放卷L_离合器rst'
  4 = 'Un_R Brake' | chinese: '放卷R_刹车' | Chinese: '放卷R_刹车'
  5 = 'Un_R Clutch Out' | chinese: '放卷R_离合器out' | Chinese: '放卷R_离合器out'
  6 = 'Un_R Clutch RST' | chinese: '放卷R_离合器rst' | Chinese: '放卷R_离合器rst'
  7 = 'Re_L Clutch Out' | chinese: '收卷L_离合器out' | Chinese: '收卷L_离合器out'
  8 = 'Re_L Clutch RST' | chinese: '收卷L_离合器rst' | Chinese: '收卷L_离合器rst'
  9 = 'Re_R Clutch Out' | chinese: '收卷R_离合器out' | Chinese: '收卷R_离合器out'
  10 = 'Re_R Clutch RST' | chinese: '收卷R_离合器rst' | Chinese: '收卷R_离合器rst'
  11 = 'S1 Drive enabled' | chinese: '导向压轮电机使能' | Chinese: '导向压轮电机使能'
  12 = 'S1 Forward/Reverse' | chinese: '导向压轮电机正/反转' | Chinese: '导向压轮电机正/反转'
  13 = 'S1_Break' | chinese: '导向压轮电机刹车' | Chinese: '导向压轮电机刹车'
  14 = ''
  15 = ''
  16 = ''
   = ''
END_TEXTLIST

// ---- VISUs/HMI_IO监控文字/EL2809_M_3.TcTLO
TEXTLIST EL2809_M_3
  1 = 'Vac Pump Run/Stop' | chinese: '真空吸附启停' | Chinese: '真空吸附启停'
  2 = 'Cylinder S2 rises' | chinese: '压辊气缸S2上升' | Chinese: '压辊气缸S2上升'
  3 = 'Cylinder S3 rises' | chinese: '压辊气缸S3上升' | Chinese: '压辊气缸S3上升'
  4 = 'Cylinder S4 rises' | chinese: '压辊气缸S4上升' | Chinese: '压辊气缸S4上升'
  5 = 'Cylinder S5 rises' | chinese: '压辊气缸S5上升' | Chinese: '压辊气缸S5上升'
  6 = 'Cylinder S6 rises' | chinese: '压辊气缸S6上升' | Chinese: '压辊气缸S6上升'
  7 = 'Cylinder S2 drops' | chinese: '压辊气缸S2下降' | Chinese: '压辊气缸S2下降'
  8 = 'Cylinder S3 drops' | chinese: '压辊气缸S3下降' | Chinese: '压辊气缸S3下降'
  9 = 'Cylinder S4 drops' | chinese: '压辊气缸S4下降' | Chinese: '压辊气缸S4下降'
  10 = 'Cylinder S5 drops' | chinese: '压辊气缸S5下降' | Chinese: '压辊气缸S5下降'
  11 = 'Cylinder S6 drops' | chinese: '压辊气缸S6下降' | Chinese: '压辊气缸S6下降'
  12 = ''
  13 = ''
  14 = ''
  15 = ''
  16 = ''
   = ''
END_TEXTLIST

// ---- VISUs/HMI_IO监控文字/EL2809_S_1.TcTLO
TEXTLIST EL2809_S_1
  1 = 'W circulation pump 1' | chinese: '二级墨盒白循环泵1' | Chinese: '二级墨盒白循环泵1'
  2 = 'W circulation pump 2' | chinese: '二级墨盒白循环泵2' | Chinese: '二级墨盒白循环泵2'
  3 = 'Purge Valve' | chinese: '正压电磁阀' | Chinese: '正压电磁阀'
  4 = 'Vacuum Valve White' | chinese: '负压电磁阀白' | Chinese: '负压电磁阀白'
  5 = 'Vacuum Valve Colcor' | chinese: '负压电磁阀彩' | Chinese: '负压电磁阀彩'
  6 = 'Test piece of power' | chinese: '探块电源' | Chinese: '探块电源'
  7 = ''
  8 = ''
  9 = ''
  10 = ''
  11 = ''
  12 = ''
  13 = ''
  14 = ''
  15 = ''
  16 = ''
   = ''
END_TEXTLIST

// ---- VISUs/HMI_IO监控文字/EL2904_M_1.TcTLO
TEXTLIST EL2904_M_1
  1 = 'Safety output 1' | chinese: '继电器输出' | Chinese: '继电器输出'
  2 = 'Safety output 2' | chinese: '继电器输出' | Chinese: '继电器输出'
  3 = 'Safety output 3' | chinese: '继电器输出' | Chinese: '继电器输出'
  4 = 'Safety output 4' | chinese: '继电器输出' | Chinese: '继电器输出'
   = ''
END_TEXTLIST

// ---- VISUs/F99_Monitor.TcVIS
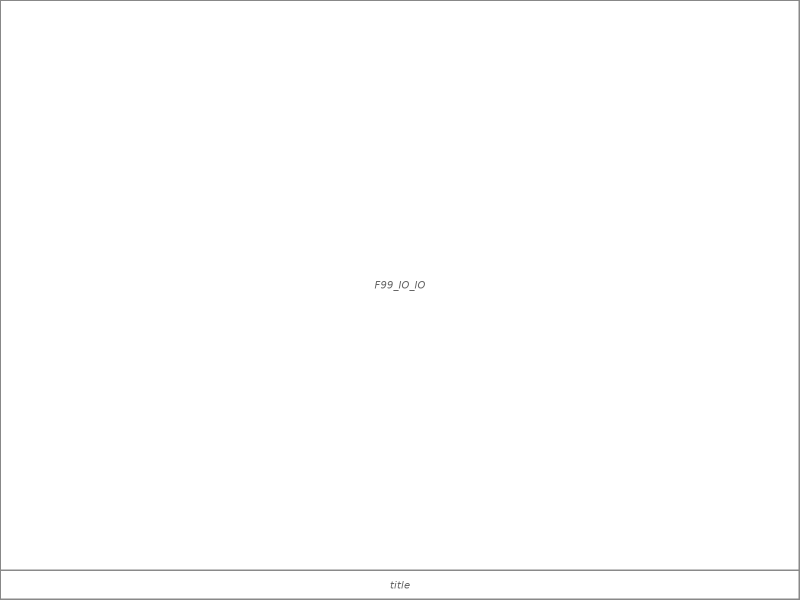
VISUALIZATION F99_Monitor  // 800x600
    Frame (0,570 800x30)
        shows title()
    TabControl (0,0 800x570)
        shows F99_IO_IO()
        shows F99_IO_IO_1()
        shows F99_IO_IO_2()
        shows F99_IO_ETHERCAT()
        shows F99_IO_SYSINFO()
        [3]: TabTitle=EtherCAT
        [4]: TabTitle=SysInfo
END_VISUALIZATION

// ---- VISUs/F4_System.TcVIS
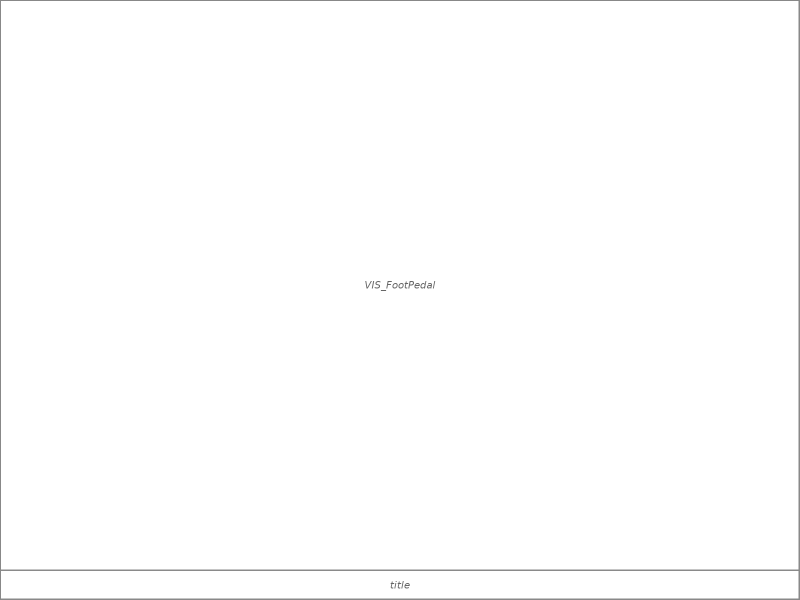
VISUALIZATION F4_System  // 800x600
    TabControl (0,0 800x570)
        shows VIS_FootPedal()
        shows VIS_SaftyGuard()
        shows VIS_SystemEnvironment()
        [0]: TabTitle=FootPedal
        [1]: TabTitle=SaftyGuard
        [2]: TabTitle=Environment
    Frame (0,570 800x30)
        shows title()
END_VISUALIZATION

// ---- VISUs/F3_MediaTransport.TcVIS
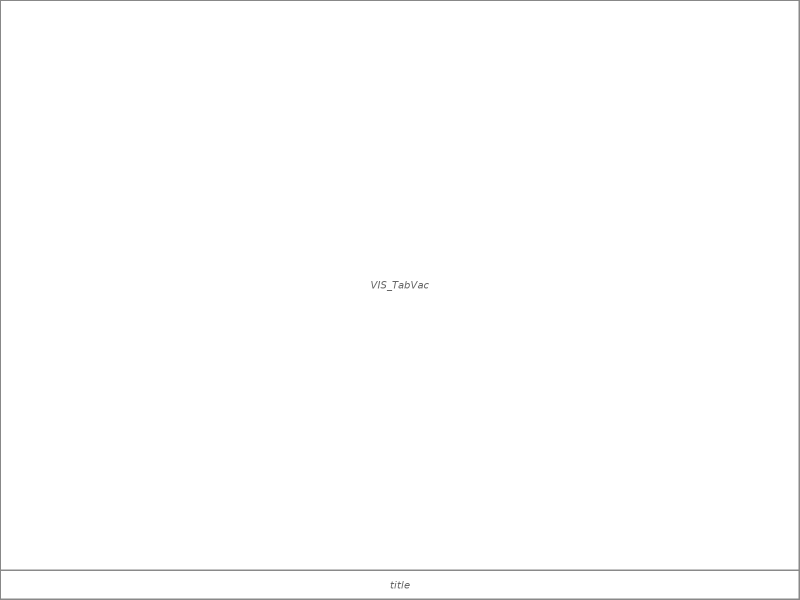
VISUALIZATION F3_MediaTransport  // 800x600
    TabControl (0,0 800x570)
        shows VIS_TabVac()
        shows VIS_UpDownSlot()
        [0]: TabTitle=TabVac
        [1]: TabTitle=UpDownSlot
    Frame (0,570 800x30)
        shows title()
END_VISUALIZATION

// ---- VISUs/F6_UVLed.TcVIS
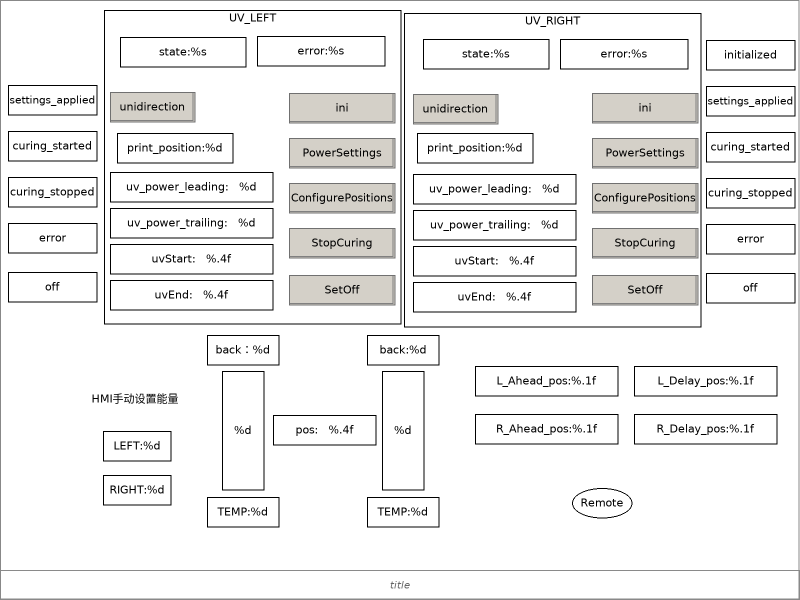
VISUALIZATION F6_UVLed  // 800x600
    RoundedRectangle (404,13 297x314), "UV_RIGHT"
    RoundedRectangle (104,10 297x314), "UV_LEFT"
    Rectangle (222,371 42x119), "%d", text variable: GVL.set_uv_power_left, colour toggle: GVL.set_uv_power_left<>0
    Rectangle (382,371 42x119), "%d", text variable: GVL.set_uv_power_right, colour toggle: GVL.set_uv_power_right<>0
    Rectangle (273,415 103x30), "pos: %.4f", text variable: Axis[1].Ref.NcToPlc.ActPos
    Button (289,93 106x30), "ini", colour toggle: GVL_API.stUVLed[1].Initialize
        toggle GVL_API.stUVLed[1].Initialize
    Rectangle (120,37 126x30), "state:%s", text list: 'TextList_UVLed_state', text index: GVL_API.stUVLed[1].state
    Rectangle (257,36 128x30), "error:%s", text list: 'TextList_UVLed_errorid', text index: GVL_API.stUVLed[1].error_code
    Rectangle (110,172 163x30), "uv_power_leading: %d", text variable: GVL_API.stUVLed[1].uv_power_leading
        OnMouseDown: write GVL_API.stUVLed[1].uv_power_leading via Default
    Button (110,92 85x30), "unidirection", colour toggle: GVL_API.stUVLed[1].unidirection
        toggle GVL_API.stUVLed[1].unidirection
    Rectangle (110,208 163x30), "uv_power_trailing: %d", text variable: GVL_API.stUVLed[1].uv_power_trailing
        OnMouseDown: write GVL_API.stUVLed[1].uv_power_trailing via Default
    Rectangle (110,244 163x30), "uvStart: %.4f", text variable: GVL_API.stUVLed[1].uvStart
        OnMouseDown: write GVL_API.stUVLed[1].uvStart via Default
    Rectangle (110,280 163x30), "uvEnd: %.4f", text variable: GVL_API.stUVLed[1].uvEnd
        OnMouseDown: write GVL_API.stUVLed[1].uvEnd via Default
    Button (289,138 106x30), "PowerSettings", colour toggle: GVL_API.stUVLed[1].ConfigurePowerSettings
        toggle GVL_API.stUVLed[1].ConfigurePowerSettings
    Button (289,275 106x30), "SetOff", colour toggle: GVL_API.stUVLed[1].SetOff
        toggle GVL_API.stUVLed[1].SetOff
    Button (289,183 106x30), "ConfigurePositions", colour toggle: GVL_API.stUVLed[1].ConfigurePositions
        toggle GVL_API.stUVLed[1].ConfigurePositions
    Button (289,228 106x30), "StopCuring", colour toggle: GVL_API.stUVLed[1].StopCuring
        toggle GVL_API.stUVLed[1].StopCuring
    Button (592,93 106x30), "ini", colour toggle: GVL_API.stUVLed[2].Initialize
        toggle GVL_API.stUVLed[2].Initialize
    Rectangle (423,39 126x30), "state:%s", text list: 'TextList_UVLed_state', text index: GVL_API.stUVLed[2].state
    Rectangle (560,39 128x30), "error:%s", text list: 'TextList_UVLed_errorid', text index: GVL_API.stUVLed[2].error_code
    Rectangle (413,174 163x30), "uv_power_leading: %d", text variable: GVL_API.stUVLed[2].uv_power_leading
        OnMouseDown: write GVL_API.stUVLed[2].uv_power_leading via Default
    Button (413,94 85x30), "unidirection", colour toggle: GVL_API.stUVLed[2].unidirection
        toggle GVL_API.stUVLed[2].unidirection
    Rectangle (413,210 163x30), "uv_power_trailing: %d", text variable: GVL_API.stUVLed[2].uv_power_trailing
        OnMouseDown: write GVL_API.stUVLed[2].uv_power_trailing via Default
    Rectangle (413,246 163x30), "uvStart: %.4f", text variable: GVL_API.stUVLed[2].uvStart
        OnMouseDown: write GVL_API.stUVLed[2].uvStart via Default
    Rectangle (413,282 163x30), "uvEnd: %.4f", text variable: GVL_API.stUVLed[2].uvEnd
        OnMouseDown: write GVL_API.stUVLed[2].uvEnd via Default
    Button (592,138 106x30), "PowerSettings", colour toggle: GVL_API.stUVLed[2].ConfigurePowerSettings
        toggle GVL_API.stUVLed[2].ConfigurePowerSettings
    Button (592,275 106x30), "SetOff", colour toggle: GVL_API.stUVLed[2].SetOff
        toggle GVL_API.stUVLed[2].SetOff
    Button (592,183 106x30), "ConfigurePositions", colour toggle: GVL_API.stUVLed[2].ConfigurePositions
        toggle GVL_API.stUVLed[2].ConfigurePositions
    Button (592,228 106x30), "StopCuring", colour toggle: GVL_API.stUVLed[2].StopCuring
        toggle GVL_API.stUVLed[2].StopCuring
    Rectangle (207,497 72x30), "TEMP:%d", text variable: GVL.HMI_TEMP_L
    Rectangle (367,497 72x30), "TEMP:%d", text variable: GVL.HMI_TEMP_R
    Rectangle (207,335 72x30), "back：%d", text variable: GVL.HMI_power_L
    Rectangle (367,335 72x30), "back:%d", text variable: GVL.HMI_power_R
    Rectangle (103,431 68x30), "LEFT:%d", text variable: PRG_SerialComm.uv_power_left_t
        OnMouseDown: toggle 
        OnMouseDown: write PRG_SerialComm.uv_power_left_t via Default
    Rectangle (103,475 68x30), "RIGHT:%d", text variable: PRG_SerialComm.uv_power_right_t
        OnMouseDown: write PRG_SerialComm.uv_power_right_t via Default
    Rectangle (417,133 116x30), "print_position:%d", text variable: GVL_API.stUVLed[2].initial_print_position
        OnMouseDown: write GVL_API.stUVLed[2].initial_print_position via Default
    Rectangle (117,133 116x30), "print_position:%d", text variable: GVL_API.stUVLed[1].initial_print_position
        OnMouseDown: write GVL_API.stUVLed[1].initial_print_position via Default
    Frame (0,570 800x30)
        shows title()
    Label (60,384 150x30), "HMI手动设置能量"
    Rectangle (475,366 143x30), "L_Ahead_pos:%.1f", text variable: GVL_API.stUVLed[1].ahead_pos
        OnMouseDown: write GVL_API.stUVLed[1].ahead_pos via Default
    Rectangle (475,414 143x30), "R_Ahead_pos:%.1f", text variable: GVL_API.stUVLed[2].ahead_pos
        OnMouseDown: write GVL_API.stUVLed[2].ahead_pos via Default
    Rectangle (634,366 143x30), "L_Delay_pos:%.1f", text variable: GVL_API.stUVLed[1].delay_pos
        OnMouseDown: write GVL_API.stUVLed[1].delay_pos via Default
    Rectangle (634,414 143x30), "R_Delay_pos:%.1f", text variable: GVL_API.stUVLed[2].delay_pos
        OnMouseDown: write GVL_API.stUVLed[2].delay_pos via Default
    Ellipse (572,488 60x30), "Remote", colour toggle: GVL.UVisRemote
    RoundedRectangle (8,85 89x30), "settings_applied", colour toggle: GVL_API.stUVLed[1].settings_applied
    RoundedRectangle (8,131 89x30), "curing_started", colour toggle: GVL_API.stUVLed[1].curing_started
    RoundedRectangle (8,223 89x30), "error", colour toggle: GVL_API.stUVLed[1].error
    RoundedRectangle (8,272 89x30), "off", colour toggle: GVL_API.stUVLed[1].off
    RoundedRectangle (8,177 89x30), "curing_stopped", colour toggle: GVL_API.stUVLed[1].curing_stopped
    RoundedRectangle (706,273 89x30), "off", colour toggle: GVL_API.stUVLed[2].off
    RoundedRectangle (706,40 89x30), "initialized", colour toggle: GVL_API.stUVLed[2].initialized
    RoundedRectangle (706,86 89x30), "settings_applied", colour toggle: GVL_API.stUVLed[2].settings_applied
    RoundedRectangle (706,132 89x30), "curing_started", colour toggle: GVL_API.stUVLed[2].curing_started
    RoundedRectangle (706,224 89x30), "error", colour toggle: GVL_API.stUVLed[2].error
    RoundedRectangle (706,178 89x30), "curing_stopped", colour toggle: GVL_API.stUVLed[2].curing_stopped
END_VISUALIZATION

// ---- VISUs/VIS文本/PLC/subinklevel.TcTLO
TEXTLIST subinklevel
  1 = 'W1'
  2 = 'W2'
  3 = 'LM1'
  4 = 'LC1'
  5 = 'Y1'
  6 = 'M1'
  7 = 'C1'
  8 = 'K1'
  9 = 'K2'
  10 = 'C2'
  11 = 'M2'
  12 = 'Y2'
  13 = 'LC2'
  14 = 'LM2'
  15 = 'W3'
  16 = 'W4'
   = ''
END_TEXTLIST

// ---- VISUs/VIS文本/PLC/TextListSpitUnitErrorid.TcTLO
TEXTLIST TextListSpitUnitErrorid
  0 = 'no_error'
  1 = 'not_connected'
  2 = 'invalid_state'
  3 = 'homing_error'
  4 = 'trigger_limit'
  5 = 'io_error'
  6 = 'unknown_error'
  666 = 'emergency_error'
  7 = 'Drive_not_ready_for_operation'
   = ''
END_TEXTLIST

// ---- VISUs/VIS文本/PLC/TextList_FootPedalerroid.TcTLO
TEXTLIST TextList_FootPedalerroid
  0 = 'no_error'
  1 = 'not_connected'
  2 = 'invalid_state'
  3 = 'io_error'
  4 = 'unknown_error'
  666 = 'emergency_error'
   = ''
END_TEXTLIST

// ---- VISUs/VIS文本/PLC/TextList_RTRstate.TcTLO
TEXTLIST TextList_RTRstate
  0 = 'off'
  1 = 'initializing'
  2 = 'ready'
  4 = 'active'
  5 = 'tensioning'
  6 = 'Tensioned_locked'
  8 = 'tensioned'
  9 = 'untensioning'
  10 = 'setting_off'
  13 = 'brake_enabled'
  100 = 'error'
   = ''
END_TEXTLIST

// ---- VISUs/VIS文本/PLC/TextList_SafetyGuarderrorid.TcTLO
TEXTLIST TextList_SafetyGuarderrorid
  0 = 'no_error'
  1 = 'not_connected'
  2 = 'invalid_state'
  4 = 'emergency_error'
  8 = 'interlock_error'
  16 = 'shuttle_crash_error'
  32 = 'limit_switch_error'
  64 = 'io_error'
  128 = 'unknown_error'
   = ''
END_TEXTLIST

// ---- VISUs/VIS文本/PLC/TextList_UVLed_errorid.TcTLO
TEXTLIST TextList_UVLed_errorid
  0 = 'no_error'
  1 = 'not_connected'
  2 = 'invalid_state'
  3 = 'unknown_error'
  666 = 'emergency_error'
   = ''
END_TEXTLIST

// ---- VISUs/VIS文本/PLC/TextList_UVLed_state.TcTLO
TEXTLIST TextList_UVLed_state
  0 = 'off'
  1 = 'initializing'
  2 = 'ready'
  3 = 'applying_settings'
  4 = 'settings_applied'
  10 = 'ready_for_curing'
  5 = 'curing'
  6 = 'setting_off'
  100 = 'error'
   = ''
END_TEXTLIST

// ---- VISUs/VIS文本/PLC/TextList_zErrorid.TcTLO
TEXTLIST TextList_zErrorid
  0 = 'no_error'
  1 = 'not_connected'
  2 = 'invalid_state'
  3 = 'homing_error'
  4 = 'cmd_timeout'
  5 = 'TBD_error'
  6 = 'io_error'
  7 = 'unknown_error'
  8 = 'actuator_out_of_pos_range'
  9 = 'actuator_out_of_neg_range'
  10 = 'homing_timeout'
  11 = 'parameter_out_of_range'
  12 = 'trigger_Limit'
  666 = 'emergency_error'
  13 = 'Drive_not_ready_for_operation'
   = ''
END_TEXTLIST

// ---- VISUs/报警/Visualization_LogEvent.TcVIS
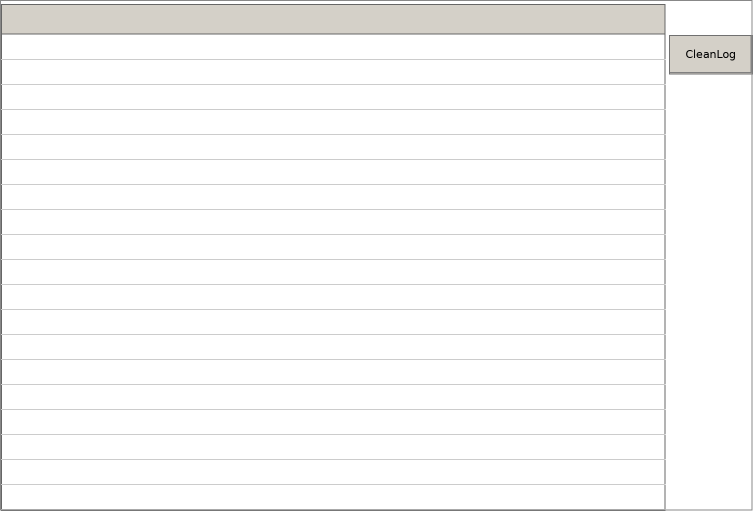
VISUALIZATION Visualization_LogEvent  // 753x511
    Button (669,35 84x39), "CleanLog"
        tap Alm_bHMIClearHistory
    Table (1,4 664x507), data array: AlarmHistoryArray
        p3854506369: AlarmHistoryArray[INDEX].EventMessage
        p1892666644: AlarmHistoryArray[INDEX].EventId
        p338671338: AlarmHistoryArray[INDEX].EventTime
END_VISUALIZATION
